LIN {X 0,Y 248.357,Z 469.454,A -85,B 0,C 180,E1 -18796.916,E2 -18796.916} C_VEL
LIN {X 0,Y 247.432,Z 473.592,A -85,B 0,C 180,E1 -18800.188,E2 -18800.188} C_VEL
LIN {X 0,Y 246.966,Z 476.493,A -85,B 0,C 180,E1 -18803.464,E2 -18803.464} C_VEL
LIN {X 0,Y 246.805,Z 478.221,A -85,B 0,C 180,E1 -18806.735,E2 -18806.735} C_VEL
LIN {X 0,Y 246.889,Z 478.812,A -85,B 0,C 180,E1 -18810,E2 -18810} C_VEL
LIN {X 0,Y 246.805,Z 478.208,A -85,B 0,C 180,E1 -18813.265,E2 -18813.265} C_VEL
LIN {X 0,Y 246.966,Z 476.463,A -85,B 0,C 180,E1 -18816.536,E2 -18816.536} C_VEL
LIN {X 0,Y 247.428,Z 473.551,A -85,B 0,C 180,E1 -18819.813,E2 -18819.813} C_VEL
LIN {X 0,Y 248.352,Z 469.403,A -85,B 0,C 180,E1 -18823.084,E2 -18823.084} C_VEL
LIN {X 0,Y 249.899,Z 463.909,A -85,B 0,C 180,E1 -18826.334,E2 -18826.334} C_VEL
LIN {X 0,Y 252.033,Z 456.92,A -85,B 0,C 180,E1 -18829.55,E2 -18829.55} C_VEL
LIN {X 0,Y 254.843,Z 448.224,A -85,B 0,C 180,E1 -18832.711,E2 -18832.711} C_VEL
LIN {X 0,Y 257.993,Z 438.986,A -85,B 0,C 180,E1 -18835.407,E2 -18835.407} C_VEL
LIN {X 0,Y 260.373,Z 431.227,A -85,B 0,C 180,E1 -18837.314,E2 -18837.314} C_VEL
LIN {X 0,Y 263.812,Z 420.385,A -85,B 0,C 180,E1 -18839.528,E2 -18839.528} C_VEL
LIN {X 0,Y 267.196,Z 408.548,A -85,B 0,C 180,E1 -18841.518,E2 -18841.518} C_VEL
LIN {X 0,Y 270.674,Z 395.599,A -85,B 0,C 180,E1 -18843.265,E2 -18843.265} C_VEL
LIN {X 0,Y 273.816,Z 381.642,A -85,B 0,C 180,E1 -18844.781,E2 -18844.781} C_VEL
LIN {X 0,Y 276.434,Z 367.299,A -85,B 0,C 180,E1 -18846.01,E2 -18846.01} C_VEL
LIN {X 0,Y 278.793,Z 352.325,A -85,B 0,C 180,E1 -18846.947,E2 -18846.947} C_VEL
LIN {X 0,Y 280.556,Z 336.654,A -85,B 0,C 180,E1 -18847.633,E2 -18847.633} C_VEL
LIN {X 0,Y 281.741,Z 316.789,A -85,B 0,C 180,E1 -18848.182,E2 -18848.182} C_VEL
LIN {X 0,Y 285.687,Z 232.335,A -85,B 0,C 180,E1 -18850.234,E2 -18850.234} C_VEL
LIN {X 0,Y 278.998,Z 217.135,A -85,B 0,C 180,E1 -18851.915,E2 -18851.915} C_VEL
LIN {X 0,Y 272.04,Z 203.261,A -85,B 0,C 180,E1 -18853.734,E2 -18853.734} C_VEL
LIN {X 0,Y 264.682,Z 190.304,A -85,B 0,C 180,E1 -18855.764,E2 -18855.764} C_VEL
LIN {X 0,Y 258.697,Z 180.792,A -85,B 0,C 180,E1 -18857.519,E2 -18857.519} C_VEL
LIN {X 0,Y 255.268,Z 175.543,A -85,B 0,C 180,E1 -18858.582,E2 -18858.582} C_VEL
LIN {X 0,Y 252.372,Z 171.249,A -85,B 0,C 180,E1 -18859.514,E2 -18859.514} C_VEL
LIN {X 0,Y 249.479,Z 166.762,A -85,B 0,C 180,E1 -18860.601,E2 -18860.601} C_VEL
LIN {X 0,Y 249.055,Z 165.14,A -85,B 0,C 180,E1 -18861.496,E2 -18861.496} C_VEL
LIN {X 0,Y 249.061,Z 165.021,A -85,B 0,C 180,E1 -18865.642,E2 -18865.642} C_VEL
LIN {X 0,Y 249.052,Z 165.043,A -85,B 0,C 180,E1 -18869.473,E2 -18869.473} C_VEL
LIN {X 0,Y 249.076,Z 165.066,A -85,B 0,C 180,E1 -18873.163,E2 -18873.163} C_VEL
LIN {X 0,Y 249.083,Z 165.081,A -85,B 0,C 180,E1 -18876.733,E2 -18876.733} C_VEL
LIN {X 0,Y 249.112,Z 165.064,A -85,B 0,C 180,E1 -18880.212,E2 -18880.212} C_VEL
LIN {X 0,Y 249.243,Z 165.041,A -85,B 0,C 180,E1 -18883.622,E2 -18883.622} C_VEL
LIN {X 0,Y 249.245,Z 165.05,A -85,B 0,C 180,E1 -18888.616,E2 -18888.616} C_VEL
LIN {X 0,Y 249.42,Z 165.025,A -85,B 0,C 180,E1 -18891.901,E2 -18891.901} C_VEL
LIN {X 0,Y 249.281,Z 165.035,A -85,B 0,C 180,E1 -18895.148,E2 -18895.148} C_VEL
LIN {X 0,Y 249.674,Z 164.998,A -85,B 0,C 180,E1 -18898.387,E2 -18898.387} C_VEL
LIN {X 0,Y 249.665,Z 164.984,A -85,B 0,C 180,E1 -18901.613,E2 -18901.613} C_VEL
LIN {X 0,Y 249.427,Z 165.032,A -85,B 0,C 180,E1 -18906.541,E2 -18906.541} C_VEL
LIN {X 0,Y 249.344,Z 165.03,A -85,B 0,C 180,E1 -18909.737,E2 -18909.737} C_VEL
LIN {X 0,Y 249.172,Z 165.046,A -85,B 0,C 180,E1 -18914.706,E2 -18914.706} C_VEL
LIN {X 0,Y 249.096,Z 165.075,A -85,B 0,C 180,E1 -18918.081,E2 -18918.081} C_VEL
LIN {X 0,Y 249.044,Z 165.074,A -85,B 0,C 180,E1 -18921.522,E2 -18921.522} C_VEL
LIN {X 0,Y 249.048,Z 165.066,A -85,B 0,C 180,E1 -18925.442,E2 -18925.442} C_VEL
LIN {X 0,Y 249.035,Z 165.064,A -85,B 0,C 180,E1 -18928.973,E2 -18928.973} C_VEL
LIN {X 0,Y 249.028,Z 165.016,A -85,B 0,C 180,E1 -18932.426,E2 -18932.426} C_VEL
LIN {X 0,Y 249.03,Z 165.093,A -85,B 0,C 180,E1 -18936.346,E2 -18936.346} C_VEL
LIN {X 0,Y 249.032,Z 165.261,A -85,B 0,C 180,E1 -18939.157,E2 -18939.157} C_VEL
LIN {X 0,Y 249.258,Z 166.289,A -85,B 0,C 180,E1 -18939.571,E2 -18939.571} C_VEL
LIN {X 0,Y 250.775,Z 168.943,A -85,B 0,C 180,E1 -18940.134,E2 -18940.134} C_VEL
LIN {X 0,Y 252.601,Z 170.697,A -85,B 0,C 180,E1 -18940.7,E2 -18940.7} C_VEL
LIN {X 0,Y 254.742,Z 174.012,A -85,B 0,C 180,E1 -18941.397,E2 -18941.397} C_VEL
LIN {X 0,Y 256.104,Z 175.59,A -85,B 0,C 180,E1 -18941.808,E2 -18941.808} C_VEL
LIN {X 0,Y 258.812,Z 179.338,A -85,B 0,C 180,E1 -18942.627,E2 -18942.627} C_VEL
LIN {X 0,Y 263.301,Z 186.225,A -85,B 0,C 180,E1 -18943.947,E2 -18943.947} C_VEL
LIN {X 0,Y 270.19,Z 197.804,A -85,B 0,C 180,E1 -18945.869,E2 -18945.869} C_VEL
LIN {X 0,Y 277.344,Z 211.184,A -85,B 0,C 180,E1 -18947.751,E2 -18947.751} C_VEL
LIN {X 0,Y 283.547,Z 224.507,A -85,B 0,C 180,E1 -18949.321,E2 -18949.321} C_VEL
LIN {X 0,Y 285.786,Z 229.616,A -85,B 0,C 180,E1 -18949.872,E2 -18949.872} C_VEL
LIN {X 0,Y 281.718,Z 316.592,A -85,B 0,C 180,E1 -18951.984,E2 -18951.984} C_VEL
LIN {X 0,Y 280.587,Z 333.873,A -85,B 0,C 180,E1 -18952.485,E2 -18952.485} C_VEL
LIN {X 0,Y 278.901,Z 349.072,A -85,B 0,C 180,E1 -18953.183,E2 -18953.183} C_VEL
LIN {X 0,Y 276.858,Z 362.663,A -85,B 0,C 180,E1 -18954.054,E2 -18954.054} C_VEL
LIN {X 0,Y 274.288,Z 376.81,A -85,B 0,C 180,E1 -18955.253,E2 -18955.253} C_VEL
LIN {X 0,Y 271.157,Z 391.075,A -85,B 0,C 180,E1 -18956.802,E2 -18956.802} C_VEL
LIN {X 0,Y 267.701,Z 404.046,A -85,B 0,C 180,E1 -18958.548,E2 -18958.548} C_VEL
LIN {X 0,Y 264.306,Z 415.889,A -85,B 0,C 180,E1 -18960.533,E2 -18960.533} C_VEL
LIN {X 0,Y 260.969,Z 426.728,A -85,B 0,C 180,E1 -18962.754,E2 -18962.754} C_VEL
LIN {X 0,Y 258.082,Z 435.921,A -85,B 0,C 180,E1 -18965.033,E2 -18965.033} C_VEL
LIN {X 0,Y 255.039,Z 444.915,A -85,B 0,C 180,E1 -18967.734,E2 -18967.734} C_VEL
LIN {X 0,Y 252.502,Z 452.369,A -85,B 0,C 180,E1 -18970.488,E2 -18970.488} C_VEL
LIN {X 0,Y 250.312,Z 459.336,A -85,B 0,C 180,E1 -18973.694,E2 -18973.694} C_VEL
LIN {X 0,Y 248.66,Z 464.811,A -85,B 0,C 180,E1 -18976.932,E2 -18976.932} C_VEL
LIN {X 0,Y 247.663,Z 468.943,A -85,B 0,C 180,E1 -18980.197,E2 -18980.197} C_VEL
LIN {X 0,Y 247.075,Z 471.845,A -85,B 0,C 180,E1 -18983.467,E2 -18983.467} C_VEL
LIN {X 0,Y 246.873,Z 473.588,A -85,B 0,C 180,E1 -18986.736,E2 -18986.736} C_VEL
LIN {X 0,Y 246.892,Z 474.196,A -85,B 0,C 180,E1 -18990,E2 -18990} C_VEL
LIN {X 0,Y 246.871,Z 473.628,A -85,B 0,C 180,E1 -18993.264,E2 -18993.264} C_VEL
LIN {X 0,Y 247.068,Z 471.936,A -85,B 0,C 180,E1 -18996.534,E2 -18996.534} C_VEL
LIN {X 0,Y 247.647,Z 469.082,A -85,B 0,C 180,E1 -18999.804,E2 -18999.804} C_VEL
LIN {X 0,Y 248.635,Z 464.997,A -85,B 0,C 180,E1 -19003.07,E2 -19003.07} C_VEL
LIN {X 0,Y 250.273,Z 459.581,A -85,B 0,C 180,E1 -19006.309,E2 -19006.309} C_VEL
LIN {X 0,Y 252.478,Z 452.682,A -85,B 0,C 180,E1 -19009.514,E2 -19009.514} C_VEL
LIN {X 0,Y 255.366,Z 444.071,A -85,B 0,C 180,E1 -19012.662,E2 -19012.662} C_VEL
LIN {X 0,Y 258.04,Z 436.329,A -85,B 0,C 180,E1 -19014.971,E2 -19014.971} C_VEL
LIN {X 0,Y 261.403,Z 425.595,A -85,B 0,C 180,E1 -19017.631,E2 -19017.631} C_VEL
LIN {X 0,Y 265.139,Z 413.53,A -85,B 0,C 180,E1 -19020.021,E2 -19020.021} C_VEL
LIN {X 0,Y 268.63,Z 401.209,A -85,B 0,C 180,E1 -19021.991,E2 -19021.991} C_VEL
LIN {X 0,Y 272.023,Z 387.612,A -85,B 0,C 180,E1 -19023.744,E2 -19023.744} C_VEL
LIN {X 0,Y 274.945,Z 374.176,A -85,B 0,C 180,E1 -19025.118,E2 -19025.118} C_VEL
LIN {X 0,Y 277.462,Z 359.466,A -85,B 0,C 180,E1 -19026.305,E2 -19026.305} C_VEL
LIN {X 0,Y 279.677,Z 343.923,A -85,B 0,C 180,E1 -19027.205,E2 -19027.205} C_VEL
LIN {X 0,Y 281.176,Z 328.456,A -85,B 0,C 180,E1 -19027.819,E2 -19027.819} C_VEL
LIN {X 0,Y 285.935,Z 229.905,A -85,B 0,C 180,E1 -19030.23,E2 -19030.23} C_VEL
LIN {X 0,Y 279.759,Z 216.163,A -85,B 0,C 180,E1 -19031.772,E2 -19031.772} C_VEL
LIN {X 0,Y 273.11,Z 203.043,A -85,B 0,C 180,E1 -19033.497,E2 -19033.497} C_VEL
LIN {X 0,Y 264.585,Z 188.119,A -85,B 0,C 180,E1 -19035.845,E2 -19035.845} C_VEL
LIN {X 0,Y 258.741,Z 179.263,A -85,B 0,C 180,E1 -19037.552,E2 -19037.552} C_VEL
LIN {X 0,Y 256.012,Z 175.393,A -85,B 0,C 180,E1 -19038.385,E2 -19038.385} C_VEL
LIN {X 0,Y 253.144,Z 171.8,A -85,B 0,C 180,E1 -19039.275,E2 -19039.275} C_VEL
LIN {X 0,Y 252.157,Z 170.153,A -85,B 0,C 180,E1 -19039.608,E2 -19039.608} C_VEL
LIN {X 0,Y 250.029,Z 167.934,A -85,B 0,C 180,E1 -19040.283,E2 -19040.283} C_VEL
LIN {X 0,Y 249.097,Z 165.61,A -85,B 0,C 180,E1 -19040.79,E2 -19040.79} C_VEL
LIN {X 0,Y 249.017,Z 165.181,A -85,B 0,C 180,E1 -19041.1,E2 -19041.1} C_VEL
LIN {X 0,Y 249.044,Z 165.038,A -85,B 0,C 180,E1 -19045.639,E2 -19045.639} C_VEL
LIN {X 0,Y 249.002,Z 165.03,A -85,B 0,C 180,E1 -19049.466,E2 -19049.466} C_VEL
LIN {X 0,Y 249.026,Z 165.083,A -85,B 0,C 180,E1 -19053.157,E2 -19053.157} C_VEL
LIN {X 0,Y 249.008,Z 165.086,A -85,B 0,C 180,E1 -19056.725,E2 -19056.725} C_VEL
LIN {X 0,Y 249.047,Z 165.064,A -85,B 0,C 180,E1 -19060.206,E2 -19060.206} C_VEL
LIN {X 0,Y 249.095,Z 165.071,A -85,B 0,C 180,E1 -19062.51,E2 -19062.51} C_VEL
LIN {X 0,Y 248.463,Z 165.153,A -85,B 0,C 180,E1 -19063.86,E2 -19063.86} C_VEL
LIN {X 0,Y 245.618,Z 165.507,A -85,B 0,C 180,E1 -19066.061,E2 -19066.061} C_VEL
LIN {X 0,Y 243.23,Z 165.808,A -85,B 0,C 180,E1 -19067.854,E2 -19067.854} C_VEL
LIN {X 0,Y 242.277,Z 165.926,A -85,B 0,C 180,E1 -19069.246,E2 -19069.246} C_VEL
LIN {X 0,Y 242.239,Z 165.92,A -85,B 0,C 180,E1 -19069.716,E2 -19069.716} C_VEL
LIN {X 0,Y 242.402,Z 165.903,A -85,B 0,C 180,E1 -19073.34,E2 -19073.34} C_VEL
LIN {X 0,Y 242.624,Z 165.86,A -85,B 0,C 180,E1 -19078.34,E2 -19078.34} C_VEL
LIN {X 0,Y 242.632,Z 165.874,A -85,B 0,C 180,E1 -19081.66,E2 -19081.66} C_VEL
LIN {X 0,Y 242.402,Z 165.914,A -85,B 0,C 180,E1 -19086.66,E2 -19086.66} C_VEL
LIN {X 0,Y 242.269,Z 165.905,A -85,B 0,C 180,E1 -19090.023,E2 -19090.023} C_VEL
LIN {X 0,Y 242.168,Z 165.92,A -85,B 0,C 180,E1 -19095.141,E2 -19095.141} C_VEL
LIN {X 0,Y 242.073,Z 165.956,A -85,B 0,C 180,E1 -19098.624,E2 -19098.624} C_VEL
LIN {X 0,Y 242.008,Z 165.948,A -85,B 0,C 180,E1 -19102.18,E2 -19102.18} C_VEL
LIN {X 0,Y 242.068,Z 165.936,A -85,B 0,C 180,E1 -19105.838,E2 -19105.838} C_VEL
LIN {X 0,Y 242.032,Z 165.938,A -85,B 0,C 180,E1 -19109.58,E2 -19109.58} C_VEL
LIN {X 0,Y 241.981,Z 165.895,A -85,B 0,C 180,E1 -19113.492,E2 -19113.492} C_VEL
LIN {X 0,Y 242.019,Z 166.117,A -85,B 0,C 180,E1 -19116.792,E2 -19116.792} C_VEL
LIN {X 0,Y 242.243,Z 167.162,A -85,B 0,C 180,E1 -19117.274,E2 -19117.274} C_VEL
LIN {X 0,Y 243.897,Z 169.988,A -85,B 0,C 180,E1 -19117.957,E2 -19117.957} C_VEL
LIN {X 0,Y 246.212,Z 172.655,A -85,B 0,C 180,E1 -19118.763,E2 -19118.763} C_VEL
LIN {X 0,Y 251.482,Z 180.476,A -85,B 0,C 180,E1 -19120.57,E2 -19120.57} C_VEL
LIN {X 0,Y 256.805,Z 188.703,A -85,B 0,C 180,E1 -19122.272,E2 -19122.272} C_VEL
LIN {X 0,Y 264.449,Z 201.618,A -85,B 0,C 180,E1 -19124.552,E2 -19124.552} C_VEL
LIN {X 0,Y 271.551,Z 215.178,A -85,B 0,C 180,E1 -19126.538,E2 -19126.538} C_VEL
LIN {X 0,Y 278.07,Z 229.34,A -85,B 0,C 180,E1 -19128.277,E2 -19128.277} C_VEL
LIN {X 0,Y 280.293,Z 234.633,A -85,B 0,C 180,E1 -19128.857,E2 -19128.857} C_VEL
LIN {X 0,Y 276.265,Z 318.148,A -85,B 0,C 180,E1 -19130.919,E2 -19130.919} C_VEL
LIN {X 0,Y 274.995,Z 337.484,A -85,B 0,C 180,E1 -19131.468,E2 -19131.468} C_VEL
LIN {X 0,Y 273.172,Z 352.844,A -85,B 0,C 180,E1 -19132.161,E2 -19132.161} C_VEL
LIN {X 0,Y 270.766,Z 367.673,A -85,B 0,C 180,E1 -19133.113,E2 -19133.113} C_VEL
LIN {X 0,Y 268.109,Z 381.58,A -85,B 0,C 180,E1 -19134.322,E2 -19134.322} C_VEL
LIN {X 0,Y 264.756,Z 395.836,A -85,B 0,C 180,E1 -19135.895,E2 -19135.895} C_VEL
LIN {X 0,Y 261.181,Z 408.699,A -85,B 0,C 180,E1 -19137.669,E2 -19137.669} C_VEL
LIN {X 0,Y 257.616,Z 420.502,A -85,B 0,C 180,E1 -19139.689,E2 -19139.689} C_VEL
LIN {X 0,Y 254.101,Z 431.316,A -85,B 0,C 180,E1 -19141.953,E2 -19141.953} C_VEL
LIN {X 0,Y 251.09,Z 440.49,A -85,B 0,C 180,E1 -19144.288,E2 -19144.288} C_VEL
LIN {X 0,Y 247.865,Z 449.488,A -85,B 0,C 180,E1 -19147.053,E2 -19147.053} C_VEL
LIN {X 0,Y 245.287,Z 456.953,A -85,B 0,C 180,E1 -19149.89,E2 -19149.89} C_VEL
LIN {X 0,Y 243.073,Z 463.916,A -85,B 0,C 180,E1 -19153.194,E2 -19153.194} C_VEL
LIN {X 0,Y 241.414,Z 469.389,A -85,B 0,C 180,E1 -19156.532,E2 -19156.532} C_VEL
LIN {X 0,Y 240.398,Z 473.526,A -85,B 0,C 180,E1 -19159.897,E2 -19159.897} C_VEL
LIN {X 0,Y 239.889,Z 476.426,A -85,B 0,C 180,E1 -19163.27,E2 -19163.27} C_VEL
LIN {X 0,Y 239.713,Z 478.155,A -85,B 0,C 180,E1 -19166.638,E2 -19166.638} C_VEL
LIN {X 0,Y 239.801,Z 478.746,A -85,B 0,C 180,E1 -19170,E2 -19170} C_VEL
LIN {X 0,Y 239.714,Z 478.141,A -85,B 0,C 180,E1 -19173.361,E2 -19173.361} C_VEL
LIN {X 0,Y 239.888,Z 476.396,A -85,B 0,C 180,E1 -19176.73,E2 -19176.73} C_VEL
LIN {X 0,Y 240.393,Z 473.483,A -85,B 0,C 180,E1 -19180.103,E2 -19180.103} C_VEL
LIN {X 0,Y 241.409,Z 469.335,A -85,B 0,C 180,E1 -19183.468,E2 -19183.468} C_VEL
LIN {X 0,Y 243.039,Z 463.841,A -85,B 0,C 180,E1 -19186.808,E2 -19186.808} C_VEL
LIN {X 0,Y 245.285,Z 456.852,A -85,B 0,C 180,E1 -19190.11,E2 -19190.11} C_VEL
LIN {X 0,Y 248.248,Z 448.155,A -85,B 0,C 180,E1 -19193.35,E2 -19193.35} C_VEL
LIN {X 0,Y 251.07,Z 440.361,A -85,B 0,C 180,E1 -19195.714,E2 -19195.714} C_VEL
LIN {X 0,Y 253.544,Z 432.629,A -85,B 0,C 180,E1 -19197.708,E2 -19197.708} C_VEL
LIN {X 0,Y 257.018,Z 422.268,A -85,B 0,C 180,E1 -19199.936,E2 -19199.936} C_VEL
LIN {X 0,Y 260.493,Z 410.827,A -85,B 0,C 180,E1 -19201.97,E2 -19201.97} C_VEL
LIN {X 0,Y 264.008,Z 398.385,A -85,B 0,C 180,E1 -19203.759,E2 -19203.759} C_VEL
LIN {X 0,Y 267.365,Z 384.748,A -85,B 0,C 180,E1 -19205.331,E2 -19205.331} C_VEL
LIN {X 0,Y 270.141,Z 370.612,A -85,B 0,C 180,E1 -19206.637,E2 -19206.637} C_VEL
LIN {X 0,Y 272.682,Z 356.046,A -85,B 0,C 180,E1 -19207.627,E2 -19207.627} C_VEL
LIN {X 0,Y 274.531,Z 341.075,A -85,B 0,C 180,E1 -19208.375,E2 -19208.375} C_VEL
LIN {X 0,Y 275.742,Z 325.627,A -85,B 0,C 180,E1 -19208.876,E2 -19208.876} C_VEL
LIN {X 0,Y 280.23,Z 235.291,A -85,B 0,C 180,E1 -19211.083,E2 -19211.083} C_VEL
LIN {X 0,Y 279.636,Z 233.207,A -85,B 0,C 180,E1 -19211.258,E2 -19211.258} C_VEL
LIN {X 0,Y 273.037,Z 218.349,A -85,B 0,C 180,E1 -19213.002,E2 -19213.002} C_VEL
LIN {X 0,Y 266.227,Z 204.956,A -85,B 0,C 180,E1 -19214.876,E2 -19214.876} C_VEL
LIN {X 0,Y 258.939,Z 192.192,A -85,B 0,C 180,E1 -19217.006,E2 -19217.006} C_VEL
LIN {X 0,Y 251.789,Z 180.975,A -85,B 0,C 180,E1 -19219.252,E2 -19219.252} C_VEL
LIN {X 0,Y 246.85,Z 173.669,A -85,B 0,C 180,E1 -19220.925,E2 -19220.925} C_VEL
LIN {X 0,Y 244.436,Z 170.507,A -85,B 0,C 180,E1 -19221.772,E2 -19221.772} C_VEL
LIN {X 0,Y 242.548,Z 167.907,A -85,B 0,C 180,E1 -19222.48,E2 -19222.48} C_VEL
LIN {X 0,Y 242.098,Z 166.534,A -85,B 0,C 180,E1 -19222.831,E2 -19222.831} C_VEL
LIN {X 0,Y 242.029,Z 165.989,A -85,B 0,C 180,E1 -19223.469,E2 -19223.469} C_VEL
LIN {X 0,Y 241.996,Z 165.892,A -85,B 0,C 180,E1 -19227.375,E2 -19227.375} C_VEL
LIN {X 0,Y 242.038,Z 165.945,A -85,B 0,C 180,E1 -19230.587,E2 -19230.587} C_VEL
LIN {X 0,Y 242.068,Z 165.936,A -85,B 0,C 180,E1 -19234.183,E2 -19234.183} C_VEL
LIN {X 0,Y 242.054,Z 165.937,A -85,B 0,C 180,E1 -19238.297,E2 -19238.297} C_VEL
LIN {X 0,Y 242.164,Z 165.926,A -85,B 0,C 180,E1 -19243.278,E2 -19243.278} C_VEL
LIN {X 0,Y 242.181,Z 165.934,A -85,B 0,C 180,E1 -19248.28,E2 -19248.28} C_VEL
LIN {X 0,Y 242.374,Z 165.898,A -85,B 0,C 180,E1 -19251.664,E2 -19251.664} C_VEL
LIN {X 0,Y 242.241,Z 165.913,A -85,B 0,C 180,E1 -19255.007,E2 -19255.007} C_VEL
LIN {X 0,Y 242.634,Z 165.873,A -85,B 0,C 180,E1 -19258.34,E2 -19258.34} C_VEL
LIN {X 0,Y 242.624,Z 165.86,A -85,B 0,C 180,E1 -19261.66,E2 -19261.66} C_VEL
LIN {X 0,Y 242.402,Z 165.904,A -85,B 0,C 180,E1 -19266.66,E2 -19266.66} C_VEL
LIN {X 0,Y 242.268,Z 165.914,A -85,B 0,C 180,E1 -19270.024,E2 -19270.024} C_VEL
LIN {X 0,Y 242.127,Z 165.925,A -85,B 0,C 180,E1 -19275.144,E2 -19275.144} C_VEL
LIN {X 0,Y 242.032,Z 165.946,A -85,B 0,C 180,E1 -19278.628,E2 -19278.628} C_VEL
LIN {X 0,Y 241.974,Z 165.965,A -85,B 0,C 180,E1 -19282.184,E2 -19282.184} C_VEL
LIN {X 0,Y 241.988,Z 165.947,A -85,B 0,C 180,E1 -19285.826,E2 -19285.826} C_VEL
LIN {X 0,Y 241.968,Z 165.925,A -85,B 0,C 180,E1 -19289.589,E2 -19289.589} C_VEL
LIN {X 0,Y 241.98,Z 165.899,A -85,B 0,C 180,E1 -19293.493,E2 -19293.493} C_VEL
LIN {X 0,Y 241.997,Z 166.189,A -85,B 0,C 180,E1 -19297.188,E2 -19297.188} C_VEL
LIN {X 0,Y 242.322,Z 167.358,A -85,B 0,C 180,E1 -19297.599,E2 -19297.599} C_VEL
LIN {X 0,Y 243.904,Z 169.99,A -85,B 0,C 180,E1 -19298.222,E2 -19298.222} C_VEL
LIN {X 0,Y 245.675,Z 171.559,A -85,B 0,C 180,E1 -19298.817,E2 -19298.817} C_VEL
LIN {X 0,Y 247.691,Z 174.793,A -85,B 0,C 180,E1 -19299.54,E2 -19299.54} C_VEL
LIN {X 0,Y 249.386,Z 176.695,A -85,B 0,C 180,E1 -19300.094,E2 -19300.094} C_VEL
LIN {X 0,Y 252.129,Z 180.413,A -85,B 0,C 180,E1 -19300.99,E2 -19300.99} C_VEL
LIN {X 0,Y 258.645,Z 189.867,A -85,B 0,C 180,E1 -19303.009,E2 -19303.009} C_VEL
LIN {X 0,Y 266.274,Z 202.948,A -85,B 0,C 180,E1 -19305.235,E2 -19305.235} C_VEL
LIN {X 0,Y 273.18,Z 216.193,A -85,B 0,C 180,E1 -19307.127,E2 -19307.127} C_VEL
LIN {X 0,Y 279.304,Z 229.585,A -85,B 0,C 180,E1 -19308.737,E2 -19308.737} C_VEL
LIN {X 0,Y 280.283,Z 231.882,A -85,B 0,C 180,E1 -19308.989,E2 -19308.989} C_VEL
LIN {X 0,Y 275.984,Z 320.258,A -85,B 0,C 180,E1 -19311.165,E2 -19311.165} C_VEL
LIN {X 0,Y 274.806,Z 336.236,A -85,B 0,C 180,E1 -19311.671,E2 -19311.671} C_VEL
LIN {X 0,Y 272.958,Z 351.434,A -85,B 0,C 180,E1 -19312.418,E2 -19312.418} C_VEL
LIN {X 0,Y 270.761,Z 364.991,A -85,B 0,C 180,E1 -19313.345,E2 -19313.345} C_VEL
LIN {X 0,Y 268.153,Z 378.46,A -85,B 0,C 180,E1 -19314.546,E2 -19314.546} C_VEL
LIN {X 0,Y 264.835,Z 392.572,A -85,B 0,C 180,E1 -19316.132,E2 -19316.132} C_VEL
LIN {X 0,Y 261.314,Z 405.288,A -85,B 0,C 180,E1 -19317.915,E2 -19317.915} C_VEL
LIN {X 0,Y 258.14,Z 415.959,A -85,B 0,C 180,E1 -19319.757,E2 -19319.757} C_VEL
LIN {X 0,Y 254.558,Z 427.003,A -85,B 0,C 180,E1 -19322.065,E2 -19322.065} C_VEL
LIN {X 0,Y 251.641,Z 435.99,A -85,B 0,C 180,E1 -19324.349,E2 -19324.349} C_VEL
LIN {X 0,Y 248.436,Z 444.984,A -85,B 0,C 180,E1 -19327.109,E2 -19327.109} C_VEL
LIN {X 0,Y 245.766,Z 452.438,A -85,B 0,C 180,E1 -19329.931,E2 -19329.931} C_VEL
LIN {X 0,Y 243.442,Z 459.405,A -85,B 0,C 180,E1 -19333.22,E2 -19333.22} C_VEL
LIN {X 0,Y 241.706,Z 464.879,A -85,B 0,C 180,E1 -19336.549,E2 -19336.549} C_VEL
LIN {X 0,Y 240.641,Z 469.01,A -85,B 0,C 180,E1 -19339.908,E2 -19339.908} C_VEL
LIN {X 0,Y 240.02,Z 471.912,A -85,B 0,C 180,E1 -19343.274,E2 -19343.274} C_VEL
LIN {X 0,Y 239.78,Z 473.655,A -85,B 0,C 180,E1 -19346.639,E2 -19346.639} C_VEL
LIN {X 0,Y 239.805,Z 474.262,A -85,B 0,C 180,E1 -19350,E2 -19350} C_VEL
LIN {X 0,Y 239.778,Z 473.694,A -85,B 0,C 180,E1 -19353.361,E2 -19353.361} C_VEL
LIN {X 0,Y 239.991,Z 472.002,A -85,B 0,C 180,E1 -19356.727,E2 -19356.727} C_VEL
LIN {X 0,Y 240.625,Z 469.148,A -85,B 0,C 180,E1 -19360.093,E2 -19360.093} C_VEL
LIN {X 0,Y 241.68,Z 465.063,A -85,B 0,C 180,E1 -19363.453,E2 -19363.453} C_VEL
LIN {X 0,Y 243.406,Z 459.647,A -85,B 0,C 180,E1 -19366.782,E2 -19366.782} C_VEL
LIN {X 0,Y 245.725,Z 452.747,A -85,B 0,C 180,E1 -19370.073,E2 -19370.073} C_VEL
LIN {X 0,Y 248.773,Z 444.136,A -85,B 0,C 180,E1 -19373.298,E2 -19373.298} C_VEL
LIN {X 0,Y 251.594,Z 436.393,A -85,B 0,C 180,E1 -19375.657,E2 -19375.657} C_VEL
LIN {X 0,Y 254.539,Z 427.283,A -85,B 0,C 180,E1 -19377.994,E2 -19377.994} C_VEL
LIN {X 0,Y 258.047,Z 416.534,A -85,B 0,C 180,E1 -19380.255,E2 -19380.255} C_VEL
LIN {X 0,Y 261.573,Z 404.801,A -85,B 0,C 180,E1 -19382.277,E2 -19382.277} C_VEL
LIN {X 0,Y 265.08,Z 391.987,A -85,B 0,C 180,E1 -19384.062,E2 -19384.062} C_VEL
LIN {X 0,Y 268.368,Z 377.986,A -85,B 0,C 180,E1 -19385.621,E2 -19385.621} C_VEL
LIN {X 0,Y 270.991,Z 364.061,A -85,B 0,C 180,E1 -19386.851,E2 -19386.851} C_VEL
LIN {X 0,Y 273.304,Z 349.398,A -85,B 0,C 180,E1 -19387.817,E2 -19387.817} C_VEL
LIN {X 0,Y 275.096,Z 334.339,A -85,B 0,C 180,E1 -19388.515,E2 -19388.515} C_VEL
LIN {X 0,Y 276.242,Z 317.3,A -85,B 0,C 180,E1 -19389.026,E2 -19389.026} C_VEL
LIN {X 0,Y 280.441,Z 232.086,A -85,B 0,C 180,E1 -19391.115,E2 -19391.115} C_VEL
LIN {X 0,Y 273.936,Z 217.64,A -85,B 0,C 180,E1 -19392.819,E2 -19392.819} C_VEL
LIN {X 0,Y 267.329,Z 204.843,A -85,B 0,C 180,E1 -19394.619,E2 -19394.619} C_VEL
LIN {X 0,Y 260.233,Z 192.503,A -85,B 0,C 180,E1 -19396.669,E2 -19396.669} C_VEL
LIN {X 0,Y 255.358,Z 184.878,A -85,B 0,C 180,E1 -19398.157,E2 -19398.157} C_VEL
LIN {X 0,Y 251.658,Z 179.888,A -85,B 0,C 180,E1 -19399.322,E2 -19399.322} C_VEL
LIN {X 0,Y 248.577,Z 175.704,A -85,B 0,C 180,E1 -19400.342,E2 -19400.342} C_VEL
LIN {X 0,Y 246.139,Z 172.52,A -85,B 0,C 180,E1 -19401.177,E2 -19401.177} C_VEL
LIN {X 0,Y 245.214,Z 171.076,A -85,B 0,C 180,E1 -19401.514,E2 -19401.514} C_VEL
LIN {X 0,Y 242.985,Z 168.8,A -85,B 0,C 180,E1 -19402.289,E2 -19402.289} C_VEL
LIN {X 0,Y 242.069,Z 166.475,A -85,B 0,C 180,E1 -19402.825,E2 -19402.825} C_VEL
LIN {X 0,Y 241.984,Z 166.006,A -85,B 0,C 180,E1 -19403.201,E2 -19403.201} C_VEL
LIN {X 0,Y 241.989,Z 165.892,A -85,B 0,C 180,E1 -19407.377,E2 -19407.377} C_VEL
LIN {X 0,Y 241.977,Z 165.925,A -85,B 0,C 180,E1 -19410.613,E2 -19410.613} C_VEL
LIN {X 0,Y 241.997,Z 165.946,A -85,B 0,C 180,E1 -19414.197,E2 -19414.197} C_VEL
LIN {X 0,Y 241.987,Z 165.956,A -85,B 0,C 180,E1 -19418.337,E2 -19418.337} C_VEL
LIN {X 0,Y 242.115,Z 165.947,A -85,B 0,C 180,E1 -19423.318,E2 -19423.318} C_VEL
LIN {X 0,Y 242.168,Z 165.945,A -85,B 0,C 180,E1 -19428.279,E2 -19428.279} C_VEL
LIN {X 0,Y 242.239,Z 165.92,A -85,B 0,C 180,E1 -19429.716,E2 -19429.716} C_VEL
LIN {X 0,Y 241.648,Z 165.992,A -85,B 0,C 180,E1 -19431.104,E2 -19431.104} C_VEL
LIN {X 0,Y 238.752,Z 166.357,A -85,B 0,C 180,E1 -19433.365,E2 -19433.365} C_VEL
LIN {X 0,Y 236.311,Z 166.668,A -85,B 0,C 180,E1 -19435.21,E2 -19435.21} C_VEL
LIN {X 0,Y 235.369,Z 166.766,A -85,B 0,C 180,E1 -19436.643,E2 -19436.643} C_VEL
LIN {X 0,Y 235.353,Z 166.764,A -85,B 0,C 180,E1 -19437.128,E2 -19437.128} C_VEL
LIN {X 0,Y 235.641,Z 166.75,A -85,B 0,C 180,E1 -19440,E2 -19440} C_VEL
LIN {X 0,Y 235.591,Z 166.749,A -85,B 0,C 180,E1 -19441.709,E2 -19441.709} C_VEL
LIN {X 0,Y 235.353,Z 166.792,A -85,B 0,C 180,E1 -19446.86,E2 -19446.86} C_VEL
LIN {X 0,Y 235.216,Z 166.784,A -85,B 0,C 180,E1 -19450.327,E2 -19450.327} C_VEL
LIN {X 0,Y 235.115,Z 166.797,A -85,B 0,C 180,E1 -19455.606,E2 -19455.606} C_VEL
LIN {X 0,Y 235.009,Z 166.827,A -85,B 0,C 180,E1 -19459.205,E2 -19459.205} C_VEL
LIN {X 0,Y 234.954,Z 166.835,A -85,B 0,C 180,E1 -19462.883,E2 -19462.883} C_VEL
LIN {X 0,Y 234.971,Z 166.821,A -85,B 0,C 180,E1 -19466.657,E2 -19466.657} C_VEL
LIN {X 0,Y 234.932,Z 166.795,A -85,B 0,C 180,E1 -19470.567,E2 -19470.567} C_VEL
LIN {X 0,Y 234.93,Z 166.903,A -85,B 0,C 180,E1 -19474.426,E2 -19474.426} C_VEL
LIN {X 0,Y 235.123,Z 167.742,A -85,B 0,C 180,E1 -19474.942,E2 -19474.942} C_VEL
LIN {X 0,Y 236.523,Z 170.439,A -85,B 0,C 180,E1 -19475.632,E2 -19475.632} C_VEL
LIN {X 0,Y 238.958,Z 172.789,A -85,B 0,C 180,E1 -19476.553,E2 -19476.553} C_VEL
LIN {X 0,Y 241.148,Z 176.081,A -85,B 0,C 180,E1 -19477.407,E2 -19477.407} C_VEL
LIN {X 0,Y 243.323,Z 178.871,A -85,B 0,C 180,E1 -19478.201,E2 -19478.201} C_VEL
LIN {X 0,Y 249.864,Z 188.597,A -85,B 0,C 180,E1 -19480.489,E2 -19480.489} C_VEL
LIN {X 0,Y 258.016,Z 202.128,A -85,B 0,C 180,E1 -19483.105,E2 -19483.105} C_VEL
LIN {X 0,Y 265.681,Z 216.498,A -85,B 0,C 180,E1 -19485.377,E2 -19485.377} C_VEL
LIN {X 0,Y 272.909,Z 232.174,A -85,B 0,C 180,E1 -19487.405,E2 -19487.405} C_VEL
LIN {X 0,Y 274.928,Z 237.032,A -85,B 0,C 180,E1 -19487.957,E2 -19487.957} C_VEL
LIN {X 0,Y 270.002,Z 331.315,A -85,B 0,C 180,E1 -19490.317,E2 -19490.317} C_VEL
LIN {X 0,Y 268.537,Z 346.332,A -85,B 0,C 180,E1 -19490.908,E2 -19490.908} C_VEL
LIN {X 0,Y 266.404,Z 360.422,A -85,B 0,C 180,E1 -19491.687,E2 -19491.687} C_VEL
LIN {X 0,Y 263.871,Z 373.981,A -85,B 0,C 180,E1 -19492.705,E2 -19492.705} C_VEL
LIN {X 0,Y 260.839,Z 388.062,A -85,B 0,C 180,E1 -19494.099,E2 -19494.099} C_VEL
LIN {X 0,Y 257.37,Z 401.208,A -85,B 0,C 180,E1 -19495.722,E2 -19495.722} C_VEL
LIN {X 0,Y 253.439,Z 414.263,A -85,B 0,C 180,E1 -19497.736,E2 -19497.736} C_VEL
LIN {X 0,Y 249.557,Z 426.077,A -85,B 0,C 180,E1 -19500.008,E2 -19500.008} C_VEL
LIN {X 0,Y 245.953,Z 436.539,A -85,B 0,C 180,E1 -19502.494,E2 -19502.494} C_VEL
LIN {X 0,Y 242.687,Z 445.744,A -85,B 0,C 180,E1 -19505.171,E2 -19505.171} C_VEL
LIN {X 0,Y 239.686,Z 453.857,A -85,B 0,C 180,E1 -19508.047,E2 -19508.047} C_VEL
LIN {X 0,Y 237.264,Z 460.567,A -85,B 0,C 180,E1 -19510.984,E2 -19510.984} C_VEL
LIN {X 0,Y 235.276,Z 466.761,A -85,B 0,C 180,E1 -19514.405,E2 -19514.405} C_VEL
LIN {X 0,Y 233.807,Z 471.551,A -85,B 0,C 180,E1 -19517.853,E2 -19517.853} C_VEL
LIN {X 0,Y 233.035,Z 475.06,A -85,B 0,C 180,E1 -19521.327,E2 -19521.327} C_VEL
LIN {X 0,Y 232.686,Z 477.368,A -85,B 0,C 180,E1 -19524.801,E2 -19524.801} C_VEL
LIN {X 0,Y 232.644,Z 478.527,A -85,B 0,C 180,E1 -19528.269,E2 -19528.269} C_VEL
LIN {X 0,Y 232.715,Z 478.679,A -85,B 0,C 180,E1 -19530,E2 -19530} C_VEL
LIN {X 0,Y 232.625,Z 478.075,A -85,B 0,C 180,E1 -19533.464,E2 -19533.464} C_VEL
LIN {X 0,Y 232.807,Z 476.329,A -85,B 0,C 180,E1 -19536.935,E2 -19536.935} C_VEL
LIN {X 0,Y 233.372,Z 473.416,A -85,B 0,C 180,E1 -19540.41,E2 -19540.41} C_VEL
LIN {X 0,Y 234.475,Z 469.268,A -85,B 0,C 180,E1 -19543.874,E2 -19543.874} C_VEL
LIN {X 0,Y 236.17,Z 463.773,A -85,B 0,C 180,E1 -19547.312,E2 -19547.312} C_VEL
LIN {X 0,Y 238.568,Z 456.783,A -85,B 0,C 180,E1 -19550.702,E2 -19550.702} C_VEL
LIN {X 0,Y 241.686,Z 448.086,A -85,B 0,C 180,E1 -19554.023,E2 -19554.023} C_VEL
LIN {X 0,Y 244.632,Z 440.292,A -85,B 0,C 180,E1 -19556.442,E2 -19556.442} C_VEL
LIN {X 0,Y 247.186,Z 432.742,A -85,B 0,C 180,E1 -19558.433,E2 -19558.433} C_VEL
LIN {X 0,Y 250.853,Z 422.199,A -85,B 0,C 180,E1 -19560.75,E2 -19560.75} C_VEL
LIN {X 0,Y 254.445,Z 410.756,A -85,B 0,C 180,E1 -19562.824,E2 -19562.824} C_VEL
LIN {X 0,Y 258.124,Z 398.314,A -85,B 0,C 180,E1 -19564.637,E2 -19564.637} C_VEL
LIN {X 0,Y 261.583,Z 384.676,A -85,B 0,C 180,E1 -19566.234,E2 -19566.234} C_VEL
LIN {X 0,Y 264.457,Z 370.538,A -85,B 0,C 180,E1 -19567.558,E2 -19567.558} C_VEL
LIN {X 0,Y 267.16,Z 355.224,A -85,B 0,C 180,E1 -19568.605,E2 -19568.605} C_VEL
LIN {X 0,Y 269.108,Z 339.919,A -85,B 0,C 180,E1 -19569.355,E2 -19569.355} C_VEL
LIN {X 0,Y 270.361,Z 323.771,A -85,B 0,C 180,E1 -19569.862,E2 -19569.862} C_VEL
LIN {X 0,Y 274.755,Z 236.769,A -85,B 0,C 180,E1 -19572.032,E2 -19572.032} C_VEL
LIN {X 0,Y 268.537,Z 222.554,A -85,B 0,C 180,E1 -19573.748,E2 -19573.748} C_VEL
LIN {X 0,Y 261.701,Z 208.95,A -85,B 0,C 180,E1 -19575.715,E2 -19575.715} C_VEL
LIN {X 0,Y 254.909,Z 196.946,A -85,B 0,C 180,E1 -19577.788,E2 -19577.788} C_VEL
LIN {X 0,Y 248.065,Z 185.969,A -85,B 0,C 180,E1 -19580.037,E2 -19580.037} C_VEL
LIN {X 0,Y 242.294,Z 177.272,A -85,B 0,C 180,E1 -19582.097,E2 -19582.097} C_VEL
LIN {X 0,Y 239.465,Z 173.763,A -85,B 0,C 180,E1 -19583.144,E2 -19583.144} C_VEL
LIN {X 0,Y 238.568,Z 172.191,A -85,B 0,C 180,E1 -19583.509,E2 -19583.509} C_VEL
LIN {X 0,Y 236.226,Z 170.01,A -85,B 0,C 180,E1 -19584.392,E2 -19584.392} C_VEL
LIN {X 0,Y 235.091,Z 167.448,A -85,B 0,C 180,E1 -19585.049,E2 -19585.049} C_VEL
LIN {X 0,Y 234.956,Z 166.853,A -85,B 0,C 180,E1 -19585.577,E2 -19585.577} C_VEL
LIN {X 0,Y 234.97,Z 166.809,A -85,B 0,C 180,E1 -19590.157,E2 -19590.157} C_VEL
LIN {X 0,Y 234.995,Z 166.816,A -85,B 0,C 180,E1 -19593.794,E2 -19593.794} C_VEL
LIN {X 0,Y 235.013,Z 166.812,A -85,B 0,C 180,E1 -19598.97,E2 -19598.97} C_VEL
LIN {X 0,Y 235.098,Z 166.808,A -85,B 0,C 180,E1 -19603.06,E2 -19603.06} C_VEL
LIN {X 0,Y 235.144,Z 166.816,A -85,B 0,C 180,E1 -19607.924,E2 -19607.924} C_VEL
LIN {X 0,Y 235.313,Z 166.774,A -85,B 0,C 180,E1 -19611.412,E2 -19611.412} C_VEL
LIN {X 0,Y 235.352,Z 166.793,A -85,B 0,C 180,E1 -19613.14,E2 -19613.14} C_VEL
LIN {X 0,Y 235.593,Z 166.748,A -85,B 0,C 180,E1 -19618.291,E2 -19618.291} C_VEL
LIN {X 0,Y 235.583,Z 166.736,A -85,B 0,C 180,E1 -19621.71,E2 -19621.71} C_VEL
LIN {X 0,Y 235.352,Z 166.777,A -85,B 0,C 180,E1 -19626.86,E2 -19626.86} C_VEL
LIN {X 0,Y 235.215,Z 166.796,A -85,B 0,C 180,E1 -19630.328,E2 -19630.328} C_VEL
LIN {X 0,Y 235.075,Z 166.807,A -85,B 0,C 180,E1 -19635.609,E2 -19635.609} C_VEL
LIN {X 0,Y 234.97,Z 166.819,A -85,B 0,C 180,E1 -19639.209,E2 -19639.209} C_VEL
LIN {X 0,Y 234.909,Z 166.849,A -85,B 0,C 180,E1 -19642.888,E2 -19642.888} C_VEL
LIN {X 0,Y 234.926,Z 166.833,A -85,B 0,C 180,E1 -19646.663,E2 -19646.663} C_VEL
LIN {X 0,Y 234.899,Z 166.784,A -85,B 0,C 180,E1 -19650.573,E2 -19650.573} C_VEL
LIN {X 0,Y 234.941,Z 166.771,A -85,B 0,C 180,E1 -19653.114,E2 -19653.114} C_VEL
LIN {X 0,Y 234.955,Z 167.09,A -85,B 0,C 180,E1 -19654.927,E2 -19654.927} C_VEL
LIN {X 0,Y 235.253,Z 168.176,A -85,B 0,C 180,E1 -19655.337,E2 -19655.337} C_VEL
LIN {X 0,Y 236.661,Z 170.658,A -85,B 0,C 180,E1 -19655.964,E2 -19655.964} C_VEL
LIN {X 0,Y 238.946,Z 172.776,A -85,B 0,C 180,E1 -19656.819,E2 -19656.819} C_VEL
LIN {X 0,Y 241.02,Z 175.97,A -85,B 0,C 180,E1 -19657.628,E2 -19657.628} C_VEL
LIN {X 0,Y 242.677,Z 177.763,A -85,B 0,C 180,E1 -19658.218,E2 -19658.218} C_VEL
LIN {X 0,Y 245.362,Z 181.428,A -85,B 0,C 180,E1 -19659.177,E2 -19659.177} C_VEL
LIN {X 0,Y 252.257,Z 191.012,A -85,B 0,C 180,E1 -19661.473,E2 -19661.473} C_VEL
LIN {X 0,Y 257.418,Z 199.259,A -85,B 0,C 180,E1 -19663.092,E2 -19663.092} C_VEL
LIN {X 0,Y 265.508,Z 213.978,A -85,B 0,C 180,E1 -19665.483,E2 -19665.483} C_VEL
LIN {X 0,Y 272.304,Z 228.181,A -85,B 0,C 180,E1 -19667.378,E2 -19667.378} C_VEL
LIN {X 0,Y 274.866,Z 234.138,A -85,B 0,C 180,E1 -19668.075,E2 -19668.075} C_VEL
LIN {X 0,Y 270.307,Z 323.557,A -85,B 0,C 180,E1 -19670.31,E2 -19670.31} C_VEL
LIN {X 0,Y 268.975,Z 339.178,A -85,B 0,C 180,E1 -19670.863,E2 -19670.863} C_VEL
LIN {X 0,Y 266.932,Z 354.204,A -85,B 0,C 180,E1 -19671.657,E2 -19671.657} C_VEL
LIN {X 0,Y 264.787,Z 366.99,A -85,B 0,C 180,E1 -19672.583,E2 -19672.583} C_VEL
LIN {X 0,Y 262.011,Z 380.394,A -85,B 0,C 180,E1 -19673.835,E2 -19673.835} C_VEL
LIN {X 0,Y 258.594,Z 394.068,A -85,B 0,C 180,E1 -19675.435,E2 -19675.435} C_VEL
LIN {X 0,Y 254.633,Z 407.692,A -85,B 0,C 180,E1 -19677.438,E2 -19677.438} C_VEL
LIN {X 0,Y 250.714,Z 419.901,A -85,B 0,C 180,E1 -19679.697,E2 -19679.697} C_VEL
LIN {X 0,Y 247.022,Z 430.92,A -85,B 0,C 180,E1 -19682.238,E2 -19682.238} C_VEL
LIN {X 0,Y 243.655,Z 440.11,A -85,B 0,C 180,E1 -19684.821,E2 -19684.821} C_VEL
LIN {X 0,Y 240.605,Z 448.4,A -85,B 0,C 180,E1 -19687.683,E2 -19687.683} C_VEL
LIN {X 0,Y 237.549,Z 456.607,A -85,B 0,C 180,E1 -19691.216,E2 -19691.216} C_VEL
LIN {X 0,Y 235.679,Z 462.386,A -85,B 0,C 180,E1 -19694.432,E2 -19694.432} C_VEL
LIN {X 0,Y 234.152,Z 467.172,A -85,B 0,C 180,E1 -19697.872,E2 -19697.872} C_VEL
LIN {X 0,Y 233.202,Z 470.677,A -85,B 0,C 180,E1 -19701.333,E2 -19701.333} C_VEL
LIN {X 0,Y 232.725,Z 473.197,A -85,B 0,C 180,E1 -19705.248,E2 -19705.248} C_VEL
LIN {X 0,Y 232.685,Z 474.171,A -85,B 0,C 180,E1 -19708.269,E2 -19708.269} C_VEL
LIN {X 0,Y 232.72,Z 474.328,A -85,B 0,C 180,E1 -19710,E2 -19710} C_VEL
LIN {X 0,Y 232.689,Z 473.76,A -85,B 0,C 180,E1 -19713.463,E2 -19713.463} C_VEL
LIN {X 0,Y 232.916,Z 472.068,A -85,B 0,C 180,E1 -19716.932,E2 -19716.932} C_VEL
LIN {X 0,Y 233.605,Z 469.214,A -85,B 0,C 180,E1 -19720.4,E2 -19720.4} C_VEL
LIN {X 0,Y 234.741,Z 465.129,A -85,B 0,C 180,E1 -19723.858,E2 -19723.858} C_VEL
LIN {X 0,Y 236.566,Z 459.712,A -85,B 0,C 180,E1 -19727.283,E2 -19727.283} C_VEL
LIN {X 0,Y 239.024,Z 452.812,A -85,B 0,C 180,E1 -19730.661,E2 -19730.661} C_VEL
LIN {X 0,Y 242.219,Z 444.201,A -85,B 0,C 180,E1 -19733.967,E2 -19733.967} C_VEL
LIN {X 0,Y 245.682,Z 435.045,A -85,B 0,C 180,E1 -19736.779,E2 -19736.779} C_VEL
LIN {X 0,Y 248.269,Z 427.347,A -85,B 0,C 180,E1 -19738.766,E2 -19738.766} C_VEL
LIN {X 0,Y 251.909,Z 416.598,A -85,B 0,C 180,E1 -19741.073,E2 -19741.073} C_VEL
LIN {X 0,Y 255.598,Z 404.864,A -85,B 0,C 180,E1 -19743.127,E2 -19743.127} C_VEL
LIN {X 0,Y 259.214,Z 392.049,A -85,B 0,C 180,E1 -19744.943,E2 -19744.943} C_VEL
LIN {X 0,Y 262.45,Z 378.847,A -85,B 0,C 180,E1 -19746.444,E2 -19746.444} C_VEL
LIN {X 0,Y 265.14,Z 365.248,A -85,B 0,C 180,E1 -19747.685,E2 -19747.685} C_VEL
LIN {X 0,Y 267.535,Z 350.977,A -85,B 0,C 180,E1 -19748.662,E2 -19748.662} C_VEL
LIN {X 0,Y 269.481,Z 335.53,A -85,B 0,C 180,E1 -19749.411,E2 -19749.411} C_VEL
LIN {X 0,Y 270.671,Z 319.131,A -85,B 0,C 180,E1 -19749.928,E2 -19749.928} C_VEL
LIN {X 0,Y 275.026,Z 234.415,A -85,B 0,C 180,E1 -19752.028,E2 -19752.028} C_VEL
LIN {X 0,Y 269.257,Z 221.523,A -85,B 0,C 180,E1 -19753.61,E2 -19753.61} C_VEL
LIN {X 0,Y 263.002,Z 209.193,A -85,B 0,C 180,E1 -19755.392,E2 -19755.392} C_VEL
LIN {X 0,Y 256.004,Z 196.856,A -85,B 0,C 180,E1 -19757.506,E2 -19757.506} C_VEL
LIN {X 0,Y 251.35,Z 189.705,A -85,B 0,C 180,E1 -19758.983,E2 -19758.983} C_VEL
LIN {X 0,Y 245.228,Z 181.294,A -85,B 0,C 180,E1 -19761.041,E2 -19761.041} C_VEL
LIN {X 0,Y 242.54,Z 177.495,A -85,B 0,C 180,E1 -19762.013,E2 -19762.013} C_VEL
LIN {X 0,Y 239.584,Z 174.019,A -85,B 0,C 180,E1 -19763.099,E2 -19763.099} C_VEL
LIN {X 0,Y 238.583,Z 172.202,A -85,B 0,C 180,E1 -19763.511,E2 -19763.511} C_VEL
LIN {X 0,Y 236.28,Z 170.16,A -85,B 0,C 180,E1 -19764.378,E2 -19764.378} C_VEL
LIN {X 0,Y 235.011,Z 167.431,A -85,B 0,C 180,E1 -19765.083,E2 -19765.083} C_VEL
LIN {X 0,Y 234.926,Z 166.885,A -85,B 0,C 180,E1 -19765.573,E2 -19765.573} C_VEL
LIN {X 0,Y 234.899,Z 166.783,A -85,B 0,C 180,E1 -19769.427,E2 -19769.427} C_VEL
LIN {X 0,Y 234.942,Z 166.828,A -85,B 0,C 180,E1 -19773.82,E2 -19773.82} C_VEL
LIN {X 0,Y 234.938,Z 166.826,A -85,B 0,C 180,E1 -19778.963,E2 -19778.963} C_VEL
LIN {X 0,Y 235.056,Z 166.83,A -85,B 0,C 180,E1 -19783.093,E2 -19783.093} C_VEL
LIN {X 0,Y 235.1,Z 166.821,A -85,B 0,C 180,E1 -19787.921,E2 -19787.921} C_VEL
LIN {X 0,Y 235.314,Z 166.77,A -85,B 0,C 180,E1 -19791.412,E2 -19791.412} C_VEL
LIN {X 0,Y 235.353,Z 166.777,A -85,B 0,C 180,E1 -19793.14,E2 -19793.14} C_VEL
LIN {X 0,Y 235.353,Z 166.764,A -85,B 0,C 180,E1 -19797.128,E2 -19797.128} C_VEL
LIN {X 0,Y 234.825,Z 166.836,A -85,B 0,C 180,E1 -19798.559,E2 -19798.559} C_VEL
LIN {X 0,Y 233.257,Z 167.047,A -85,B 0,C 180,E1 -19799.964,E2 -19799.964} C_VEL
LIN {X 0,Y 229.377,Z 167.518,A -85,B 0,C 180,E1 -19802.792,E2 -19802.792} C_VEL
LIN {X 0,Y 228.256,Z 167.648,A -85,B 0,C 180,E1 -19804.272,E2 -19804.272} C_VEL
LIN {X 0,Y 228.16,Z 167.663,A -85,B 0,C 180,E1 -19804.775,E2 -19804.775} C_VEL
LIN {X 0,Y 228.305,Z 167.668,A -85,B 0,C 180,E1 -19807.073,E2 -19807.073} C_VEL
LIN {X 0,Y 228.151,Z 167.666,A -85,B 0,C 180,E1 -19810.651,E2 -19810.651} C_VEL
LIN {X 0,Y 228.066,Z 167.681,A -85,B 0,C 180,E1 -19814.272,E2 -19814.272} C_VEL
LIN {X 0,Y 228.004,Z 167.707,A -85,B 0,C 180,E1 -19817.953,E2 -19817.953} C_VEL
LIN {X 0,Y 227.918,Z 167.703,A -85,B 0,C 180,E1 -19822.321,E2 -19822.321} C_VEL
LIN {X 0,Y 227.944,Z 167.695,A -85,B 0,C 180,E1 -19826.602,E2 -19826.602} C_VEL
LIN {X 0,Y 227.91,Z 167.673,A -85,B 0,C 180,E1 -19830.296,E2 -19830.296} C_VEL
LIN {X 0,Y 227.908,Z 167.817,A -85,B 0,C 180,E1 -19831.876,E2 -19831.876} C_VEL
LIN {X 0,Y 228.128,Z 168.684,A -85,B 0,C 180,E1 -19832.428,E2 -19832.428} C_VEL
LIN {X 0,Y 229.574,Z 171.417,A -85,B 0,C 180,E1 -19833.195,E2 -19833.195} C_VEL
LIN {X 0,Y 232.003,Z 173.573,A -85,B 0,C 180,E1 -19834.215,E2 -19834.215} C_VEL
LIN {X 0,Y 234.076,Z 176.798,A -85,B 0,C 180,E1 -19835.122,E2 -19835.122} C_VEL
LIN {X 0,Y 236.037,Z 178.816,A -85,B 0,C 180,E1 -19835.895,E2 -19835.895} C_VEL
LIN {X 0,Y 238.662,Z 182.481,A -85,B 0,C 180,E1 -19836.935,E2 -19836.935} C_VEL
LIN {X 0,Y 241.002,Z 185.733,A -85,B 0,C 180,E1 -19837.823,E2 -19837.823} C_VEL
LIN {X 0,Y 247.459,Z 195.794,A -85,B 0,C 180,E1 -19840.151,E2 -19840.151} C_VEL
LIN {X 0,Y 254.403,Z 207.643,A -85,B 0,C 180,E1 -19842.456,E2 -19842.456} C_VEL
LIN {X 0,Y 261.667,Z 221.535,A -85,B 0,C 180,E1 -19844.697,E2 -19844.697} C_VEL
LIN {X 0,Y 268.399,Z 236.425,A -85,B 0,C 180,E1 -19846.668,E2 -19846.668} C_VEL
LIN {X 0,Y 269.564,Z 239.194,A -85,B 0,C 180,E1 -19846.999,E2 -19846.999} C_VEL
LIN {X 0,Y 264.589,Z 331.267,A -85,B 0,C 180,E1 -19849.338,E2 -19849.338} C_VEL
LIN {X 0,Y 263.073,Z 346.276,A -85,B 0,C 180,E1 -19849.934,E2 -19849.934} C_VEL
LIN {X 0,Y 260.881,Z 360.364,A -85,B 0,C 180,E1 -19850.722,E2 -19850.722} C_VEL
LIN {X 0,Y 257.941,Z 375.409,A -85,B 0,C 180,E1 -19851.88,E2 -19851.88} C_VEL
LIN {X 0,Y 254.871,Z 388.945,A -85,B 0,C 180,E1 -19853.269,E2 -19853.269} C_VEL
LIN {X 0,Y 251.148,Z 402.437,A -85,B 0,C 180,E1 -19854.994,E2 -19854.994} C_VEL
LIN {X 0,Y 247.082,Z 415.27,A -85,B 0,C 180,E1 -19857.044,E2 -19857.044} C_VEL
LIN {X 0,Y 243.407,Z 426.013,A -85,B 0,C 180,E1 -19859.169,E2 -19859.169} C_VEL
LIN {X 0,Y 239.932,Z 435.69,A -85,B 0,C 180,E1 -19861.491,E2 -19861.491} C_VEL
LIN {X 0,Y 236.231,Z 445.679,A -85,B 0,C 180,E1 -19864.444,E2 -19864.444} C_VEL
LIN {X 0,Y 233.054,Z 453.792,A -85,B 0,C 180,E1 -19867.388,E2 -19867.388} C_VEL
LIN {X 0,Y 229.973,Z 461.906,A -85,B 0,C 180,E1 -19871.134,E2 -19871.134} C_VEL
LIN {X 0,Y 227.954,Z 468.011,A -85,B 0,C 180,E1 -19874.807,E2 -19874.807} C_VEL
LIN {X 0,Y 226.814,Z 471.485,A -85,B 0,C 180,E1 -19877.473,E2 -19877.473} C_VEL
LIN {X 0,Y 225.98,Z 474.994,A -85,B 0,C 180,E1 -19881.054,E2 -19881.054} C_VEL
LIN {X 0,Y 225.589,Z 477.301,A -85,B 0,C 180,E1 -19884.637,E2 -19884.637} C_VEL
LIN {X 0,Y 225.544,Z 478.46,A -85,B 0,C 180,E1 -19888.214,E2 -19888.214} C_VEL
LIN {X 0,Y 225.631,Z 478.613,A -85,B 0,C 180,E1 -19890,E2 -19890} C_VEL
LIN {X 0,Y 225.521,Z 478.008,A -85,B 0,C 180,E1 -19893.573,E2 -19893.573} C_VEL
LIN {X 0,Y 225.734,Z 476.262,A -85,B 0,C 180,E1 -19897.154,E2 -19897.154} C_VEL
LIN {X 0,Y 226.33,Z 473.348,A -85,B 0,C 180,E1 -19900.738,E2 -19900.738} C_VEL
LIN {X 0,Y 227.552,Z 469.2,A -85,B 0,C 180,E1 -19904.305,E2 -19904.305} C_VEL
LIN {X 0,Y 229.325,Z 463.705,A -85,B 0,C 180,E1 -19907.846,E2 -19907.846} C_VEL
LIN {X 0,Y 231.892,Z 456.715,A -85,B 0,C 180,E1 -19911.327,E2 -19911.327} C_VEL
LIN {X 0,Y 235.171,Z 448.018,A -85,B 0,C 180,E1 -19914.733,E2 -19914.733} C_VEL
LIN {X 0,Y 238.225,Z 440.223,A -85,B 0,C 180,E1 -19917.211,E2 -19917.211} C_VEL
LIN {X 0,Y 240.924,Z 432.651,A -85,B 0,C 180,E1 -19919.249,E2 -19919.249} C_VEL
LIN {X 0,Y 244.736,Z 422.129,A -85,B 0,C 180,E1 -19921.606,E2 -19921.606} C_VEL
LIN {X 0,Y 248.492,Z 410.686,A -85,B 0,C 180,E1 -19923.714,E2 -19923.714} C_VEL
LIN {X 0,Y 252.297,Z 398.243,A -85,B 0,C 180,E1 -19925.556,E2 -19925.556} C_VEL
LIN {X 0,Y 255.857,Z 384.604,A -85,B 0,C 180,E1 -19927.179,E2 -19927.179} C_VEL
LIN {X 0,Y 258.862,Z 370.465,A -85,B 0,C 180,E1 -19928.517,E2 -19928.517} C_VEL
LIN {X 0,Y 261.547,Z 355.896,A -85,B 0,C 180,E1 -19929.532,E2 -19929.532} C_VEL
LIN {X 0,Y 263.557,Z 340.919,A -85,B 0,C 180,E1 -19930.289,E2 -19930.289} C_VEL
LIN {X 0,Y 264.85,Z 325.456,A -85,B 0,C 180,E1 -19930.802,E2 -19930.802} C_VEL
LIN {X 0,Y 269.474,Z 239.745,A -85,B 0,C 180,E1 -19932.943,E2 -19932.943} C_VEL
LIN {X 0,Y 268.557,Z 236.934,A -85,B 0,C 180,E1 -19933.226,E2 -19933.226} C_VEL
LIN {X 0,Y 261.412,Z 221.049,A -85,B 0,C 180,E1 -19935.315,E2 -19935.315} C_VEL
LIN {X 0,Y 253.623,Z 206.261,A -85,B 0,C 180,E1 -19937.723,E2 -19937.723} C_VEL
LIN {X 0,Y 245.542,Z 192.688,A -85,B 0,C 180,E1 -19940.44,E2 -19940.44} C_VEL
LIN {X 0,Y 238.977,Z 182.79,A -85,B 0,C 180,E1 -19942.858,E2 -19942.858} C_VEL
LIN {X 0,Y 236.193,Z 179.133,A -85,B 0,C 180,E1 -19943.94,E2 -19943.94} C_VEL
LIN {X 0,Y 235.112,Z 177.824,A -85,B 0,C 180,E1 -19944.369,E2 -19944.369} C_VEL
LIN {X 0,Y 232.676,Z 174.788,A -85,B 0,C 180,E1 -19945.373,E2 -19945.373} C_VEL
LIN {X 0,Y 231.607,Z 173.072,A -85,B 0,C 180,E1 -19945.849,E2 -19945.849} C_VEL
LIN {X 0,Y 229.286,Z 171.05,A -85,B 0,C 180,E1 -19946.824,E2 -19946.824} C_VEL
LIN {X 0,Y 228.031,Z 168.267,A -85,B 0,C 180,E1 -19947.622,E2 -19947.622} C_VEL
LIN {X 0,Y 227.873,Z 167.7,A -85,B 0,C 180,E1 -19948.379,E2 -19948.379} C_VEL
LIN {X 0,Y 227.888,Z 167.71,A -85,B 0,C 180,E1 -19952.446,E2 -19952.446} C_VEL
LIN {X 0,Y 227.916,Z 167.721,A -85,B 0,C 180,E1 -19956.368,E2 -19956.368} C_VEL
LIN {X 0,Y 227.944,Z 167.698,A -85,B 0,C 180,E1 -19960.175,E2 -19960.175} C_VEL
LIN {X 0,Y 228.059,Z 167.677,A -85,B 0,C 180,E1 -19963.898,E2 -19963.898} C_VEL
LIN {X 0,Y 228.092,Z 167.699,A -85,B 0,C 180,E1 -19967.545,E2 -19967.545} C_VEL
LIN {X 0,Y 228.254,Z 167.651,A -85,B 0,C 180,E1 -19971.144,E2 -19971.144} C_VEL
LIN {X 0,Y 228.304,Z 167.668,A -85,B 0,C 180,E1 -19972.927,E2 -19972.927} C_VEL
LIN {X 0,Y 228.552,Z 167.623,A -85,B 0,C 180,E1 -19978.238,E2 -19978.238} C_VEL
LIN {X 0,Y 228.541,Z 167.612,A -85,B 0,C 180,E1 -19981.762,E2 -19981.762} C_VEL
LIN {X 0,Y 228.304,Z 167.651,A -85,B 0,C 180,E1 -19987.073,E2 -19987.073} C_VEL
LIN {X 0,Y 228.146,Z 167.681,A -85,B 0,C 180,E1 -19990.651,E2 -19990.651} C_VEL
LIN {X 0,Y 228.042,Z 167.677,A -85,B 0,C 180,E1 -19994.274,E2 -19994.274} C_VEL
LIN {X 0,Y 227.931,Z 167.711,A -85,B 0,C 180,E1 -19997.959,E2 -19997.959} C_VEL
LIN {X 0,Y 227.89,Z 167.72,A -85,B 0,C 180,E1 -20002.304,E2 -20002.304} C_VEL
LIN {X 0,Y 227.904,Z 167.707,A -85,B 0,C 180,E1 -20006.583,E2 -20006.583} C_VEL
LIN {X 0,Y 227.873,Z 167.662,A -85,B 0,C 180,E1 -20010.28,E2 -20010.28} C_VEL
LIN {X 0,Y 227.936,Z 167.985,A -85,B 0,C 180,E1 -20012.328,E2 -20012.328} C_VEL
LIN {X 0,Y 228.225,Z 169.03,A -85,B 0,C 180,E1 -20012.806,E2 -20012.806} C_VEL
LIN {X 0,Y 229.822,Z 171.751,A -85,B 0,C 180,E1 -20013.595,E2 -20013.595} C_VEL
LIN {X 0,Y 231.973,Z 173.519,A -85,B 0,C 180,E1 -20014.484,E2 -20014.484} C_VEL
LIN {X 0,Y 234.025,Z 176.791,A -85,B 0,C 180,E1 -20015.381,E2 -20015.381} C_VEL
LIN {X 0,Y 236.113,Z 178.984,A -85,B 0,C 180,E1 -20016.202,E2 -20016.202} C_VEL
LIN {X 0,Y 238.535,Z 182.347,A -85,B 0,C 180,E1 -20017.157,E2 -20017.157} C_VEL
LIN {X 0,Y 239.835,Z 184.027,A -85,B 0,C 180,E1 -20017.647,E2 -20017.647} C_VEL
LIN {X 0,Y 243.466,Z 188.97,A -85,B 0,C 180,E1 -20018.973,E2 -20018.973} C_VEL
LIN {X 0,Y 249.488,Z 197.605,A -85,B 0,C 180,E1 -20021.03,E2 -20021.03} C_VEL
LIN {X 0,Y 254.896,Z 206.591,A -85,B 0,C 180,E1 -20022.78,E2 -20022.78} C_VEL
LIN {X 0,Y 262.69,Z 221.359,A -85,B 0,C 180,E1 -20025.153,E2 -20025.153} C_VEL
LIN {X 0,Y 269.07,Z 235.449,A -85,B 0,C 180,E1 -20027,E2 -20027} C_VEL
LIN {X 0,Y 269.494,Z 236.43,A -85,B 0,C 180,E1 -20027.119,E2 -20027.119} C_VEL
LIN {X 0,Y 265.308,Z 316.862,A -85,B 0,C 180,E1 -20029.158,E2 -20029.158} C_VEL
LIN {X 0,Y 264.038,Z 334.117,A -85,B 0,C 180,E1 -20029.674,E2 -20029.674} C_VEL
LIN {X 0,Y 262.181,Z 349.302,A -85,B 0,C 180,E1 -20030.396,E2 -20030.396} C_VEL
LIN {X 0,Y 259.683,Z 364.012,A -85,B 0,C 180,E1 -20031.38,E2 -20031.38} C_VEL
LIN {X 0,Y 256.812,Z 378.2,A -85,B 0,C 180,E1 -20032.666,E2 -20032.666} C_VEL
LIN {X 0,Y 253.561,Z 391.289,A -85,B 0,C 180,E1 -20034.16,E2 -20034.16} C_VEL
LIN {X 0,Y 249.763,Z 404.257,A -85,B 0,C 180,E1 -20035.996,E2 -20035.996} C_VEL
LIN {X 0,Y 245.944,Z 416.098,A -85,B 0,C 180,E1 -20038.086,E2 -20038.086} C_VEL
LIN {X 0,Y 242.131,Z 426.936,A -85,B 0,C 180,E1 -20040.433,E2 -20040.433} C_VEL
LIN {X 0,Y 238.319,Z 437.478,A -85,B 0,C 180,E1 -20043.274,E2 -20043.274} C_VEL
LIN {X 0,Y 234.877,Z 446.243,A -85,B 0,C 180,E1 -20046.175,E2 -20046.175} C_VEL
LIN {X 0,Y 232.388,Z 452.575,A -85,B 0,C 180,E1 -20048.721,E2 -20048.721} C_VEL
LIN {X 0,Y 229.782,Z 459.541,A -85,B 0,C 180,E1 -20052.19,E2 -20052.19} C_VEL
LIN {X 0,Y 227.846,Z 465.015,A -85,B 0,C 180,E1 -20055.714,E2 -20055.714} C_VEL
LIN {X 0,Y 226.615,Z 469.145,A -85,B 0,C 180,E1 -20059.276,E2 -20059.276} C_VEL
LIN {X 0,Y 225.886,Z 472.046,A -85,B 0,C 180,E1 -20062.851,E2 -20062.851} C_VEL
LIN {X 0,Y 225.604,Z 473.788,A -85,B 0,C 180,E1 -20066.428,E2 -20066.428} C_VEL
LIN {X 0,Y 225.636,Z 474.394,A -85,B 0,C 180,E1 -20070,E2 -20070} C_VEL
LIN {X 0,Y 225.602,Z 473.826,A -85,B 0,C 180,E1 -20073.572,E2 -20073.572} C_VEL
LIN {X 0,Y 225.841,Z 472.135,A -85,B 0,C 180,E1 -20077.151,E2 -20077.151} C_VEL
LIN {X 0,Y 226.585,Z 469.28,A -85,B 0,C 180,E1 -20080.726,E2 -20080.726} C_VEL
LIN {X 0,Y 227.821,Z 465.194,A -85,B 0,C 180,E1 -20084.288,E2 -20084.288} C_VEL
LIN {X 0,Y 229.756,Z 459.778,A -85,B 0,C 180,E1 -20087.812,E2 -20087.812} C_VEL
LIN {X 0,Y 232.353,Z 452.877,A -85,B 0,C 180,E1 -20091.283,E2 -20091.283} C_VEL
LIN {X 0,Y 235.688,Z 444.265,A -85,B 0,C 180,E1 -20094.675,E2 -20094.675} C_VEL
LIN {X 0,Y 239.312,Z 435.109,A -85,B 0,C 180,E1 -20097.551,E2 -20097.551} C_VEL
LIN {X 0,Y 242.025,Z 427.411,A -85,B 0,C 180,E1 -20099.581,E2 -20099.581} C_VEL
LIN {X 0,Y 245.84,Z 416.661,A -85,B 0,C 180,E1 -20101.93,E2 -20101.93} C_VEL
LIN {X 0,Y 249.68,Z 404.926,A -85,B 0,C 180,E1 -20104.017,E2 -20104.017} C_VEL
LIN {X 0,Y 253.411,Z 392.111,A -85,B 0,C 180,E1 -20105.865,E2 -20105.865} C_VEL
LIN {X 0,Y 256.884,Z 378.356,A -85,B 0,C 180,E1 -20107.443,E2 -20107.443} C_VEL
LIN {X 0,Y 259.776,Z 364.178,A -85,B 0,C 180,E1 -20108.728,E2 -20108.728} C_VEL
LIN {X 0,Y 262.249,Z 349.51,A -85,B 0,C 180,E1 -20109.717,E2 -20109.717} C_VEL
LIN {X 0,Y 264.15,Z 334.441,A -85,B 0,C 180,E1 -20110.431,E2 -20110.431} C_VEL
LIN {X 0,Y 265.389,Z 317.385,A -85,B 0,C 180,E1 -20110.952,E2 -20110.952} C_VEL
LIN {X 0,Y 269.656,Z 236.738,A -85,B 0,C 180,E1 -20112.984,E2 -20112.984} C_VEL
LIN {X 0,Y 264.604,Z 225.328,A -85,B 0,C 180,E1 -20114.437,E2 -20114.437} C_VEL
LIN {X 0,Y 258.537,Z 213.207,A -85,B 0,C 180,E1 -20116.248,E2 -20116.248} C_VEL
LIN {X 0,Y 251.61,Z 200.885,A -85,B 0,C 180,E1 -20118.441,E2 -20118.441} C_VEL
LIN {X 0,Y 246.873,Z 193.767,A -85,B 0,C 180,E1 -20120.013,E2 -20120.013} C_VEL
LIN {X 0,Y 241.828,Z 186.705,A -85,B 0,C 180,E1 -20121.794,E2 -20121.794} C_VEL
LIN {X 0,Y 238.628,Z 182.422,A -85,B 0,C 180,E1 -20122.992,E2 -20122.992} C_VEL
LIN {X 0,Y 236.028,Z 178.866,A -85,B 0,C 180,E1 -20124.019,E2 -20124.019} C_VEL
LIN {X 0,Y 232.804,Z 175.1,A -85,B 0,C 180,E1 -20125.329,E2 -20125.329} C_VEL
LIN {X 0,Y 231.64,Z 173.121,A -85,B 0,C 180,E1 -20125.855,E2 -20125.855} C_VEL
LIN {X 0,Y 229.208,Z 170.929,A -85,B 0,C 180,E1 -20126.886,E2 -20126.886} C_VEL
LIN {X 0,Y 228.024,Z 168.393,A -85,B 0,C 180,E1 -20127.621,E2 -20127.621} C_VEL
LIN {X 0,Y 227.857,Z 167.728,A -85,B 0,C 180,E1 -20128.376,E2 -20128.376} C_VEL
LIN {X 0,Y 227.846,Z 167.73,A -85,B 0,C 180,E1 -20132.44,E2 -20132.44} C_VEL
LIN {X 0,Y 227.858,Z 167.713,A -85,B 0,C 180,E1 -20136.361,E2 -20136.361} C_VEL
LIN {X 0,Y 227.892,Z 167.697,A -85,B 0,C 180,E1 -20140.17,E2 -20140.17} C_VEL
LIN {X 0,Y 228.019,Z 167.692,A -85,B 0,C 180,E1 -20143.895,E2 -20143.895} C_VEL
LIN {X 0,Y 228.144,Z 167.683,A -85,B 0,C 180,E1 -20149.349,E2 -20149.349} C_VEL
LIN {X 0,Y 228.305,Z 167.651,A -85,B 0,C 180,E1 -20152.927,E2 -20152.927} C_VEL
LIN {X 0,Y 228.541,Z 167.612,A -85,B 0,C 180,E1 -20158.238,E2 -20158.238} C_VEL
LIN {X 0,Y 228.55,Z 167.624,A -85,B 0,C 180,E1 -20161.762,E2 -20161.762} C_VEL
LIN {X 0,Y 228.16,Z 167.663,A -85,B 0,C 180,E1 -20164.775,E2 -20164.775} C_VEL
LIN {X 0,Y 227.466,Z 167.771,A -85,B 0,C 180,E1 -20166.251,E2 -20166.251} C_VEL
LIN {X 0,Y 224.568,Z 168.115,A -85,B 0,C 180,E1 -20168.657,E2 -20168.657} C_VEL
LIN {X 0,Y 222.125,Z 168.417,A -85,B 0,C 180,E1 -20170.621,E2 -20170.621} C_VEL
LIN {X 0,Y 221.096,Z 168.566,A -85,B 0,C 180,E1 -20172.147,E2 -20172.147} C_VEL
LIN {X 0,Y 221.022,Z 168.575,A -85,B 0,C 180,E1 -20172.664,E2 -20172.664} C_VEL
LIN {X 0,Y 220.986,Z 168.571,A -85,B 0,C 180,E1 -20177.428,E2 -20177.428} C_VEL
LIN {X 0,Y 220.886,Z 168.582,A -85,B 0,C 180,E1 -20182.675,E2 -20182.675} C_VEL
LIN {X 0,Y 220.887,Z 168.577,A -85,B 0,C 180,E1 -20187.015,E2 -20187.015} C_VEL
LIN {X 0,Y 220.878,Z 168.838,A -85,B 0,C 180,E1 -20189.027,E2 -20189.027} C_VEL
LIN {X 0,Y 221.171,Z 169.829,A -85,B 0,C 180,E1 -20189.572,E2 -20189.572} C_VEL
LIN {X 0,Y 222.599,Z 172.399,A -85,B 0,C 180,E1 -20190.407,E2 -20190.407} C_VEL
LIN {X 0,Y 225.212,Z 174.501,A -85,B 0,C 180,E1 -20191.645,E2 -20191.645} C_VEL
LIN {X 0,Y 227.136,Z 177.655,A -85,B 0,C 180,E1 -20192.604,E2 -20192.604} C_VEL
LIN {X 0,Y 229.339,Z 179.856,A -85,B 0,C 180,E1 -20193.575,E2 -20193.575} C_VEL
LIN {X 0,Y 231.995,Z 183.492,A -85,B 0,C 180,E1 -20194.743,E2 -20194.743} C_VEL
LIN {X 0,Y 233.434,Z 185.237,A -85,B 0,C 180,E1 -20195.339,E2 -20195.339} C_VEL
LIN {X 0,Y 237.5,Z 190.829,A -85,B 0,C 180,E1 -20196.974,E2 -20196.974} C_VEL
LIN {X 0,Y 243.704,Z 200.688,A -85,B 0,C 180,E1 -20199.318,E2 -20199.318} C_VEL
LIN {X 0,Y 250.45,Z 212.384,A -85,B 0,C 180,E1 -20201.66,E2 -20201.66} C_VEL
LIN {X 0,Y 257.361,Z 225.829,A -85,B 0,C 180,E1 -20203.891,E2 -20203.891} C_VEL
LIN {X 0,Y 263.792,Z 240.324,A -85,B 0,C 180,E1 -20205.863,E2 -20205.863} C_VEL
LIN {X 0,Y 264.285,Z 241.935,A -85,B 0,C 180,E1 -20206.026,E2 -20206.026} C_VEL
LIN {X 0,Y 259.243,Z 331.219,A -85,B 0,C 180,E1 -20208.315,E2 -20208.315} C_VEL
LIN {X 0,Y 257.688,Z 346.221,A -85,B 0,C 180,E1 -20208.92,E2 -20208.92} C_VEL
LIN {X 0,Y 255.427,Z 360.305,A -85,B 0,C 180,E1 -20209.714,E2 -20209.714} C_VEL
LIN {X 0,Y 252.69,Z 373.856,A -85,B 0,C 180,E1 -20210.747,E2 -20210.747} C_VEL
LIN {X 0,Y 249.267,Z 388.632,A -85,B 0,C 180,E1 -20212.261,E2 -20212.261} C_VEL
LIN {X 0,Y 245.34,Z 402.374,A -85,B 0,C 180,E1 -20214.038,E2 -20214.038} C_VEL
LIN {X 0,Y 241.145,Z 415.206,A -85,B 0,C 180,E1 -20216.125,E2 -20216.125} C_VEL
LIN {X 0,Y 237.299,Z 425.949,A -85,B 0,C 180,E1 -20218.285,E2 -20218.285} C_VEL
LIN {X 0,Y 233.454,Z 436.19,A -85,B 0,C 180,E1 -20220.812,E2 -20220.812} C_VEL
LIN {X 0,Y 229.811,Z 445.614,A -85,B 0,C 180,E1 -20223.677,E2 -20223.677} C_VEL
LIN {X 0,Y 226.454,Z 453.726,A -85,B 0,C 180,E1 -20226.69,E2 -20226.69} C_VEL
LIN {X 0,Y 223.772,Z 460.436,A -85,B 0,C 180,E1 -20229.789,E2 -20229.789} C_VEL
LIN {X 0,Y 221.491,Z 466.63,A -85,B 0,C 180,E1 -20233.407,E2 -20233.407} C_VEL
LIN {X 0,Y 219.839,Z 471.419,A -85,B 0,C 180,E1 -20237.069,E2 -20237.069} C_VEL
LIN {X 0,Y 218.941,Z 474.928,A -85,B 0,C 180,E1 -20240.764,E2 -20240.764} C_VEL
LIN {X 0,Y 218.5,Z 477.235,A -85,B 0,C 180,E1 -20244.463,E2 -20244.463} C_VEL
LIN {X 0,Y 218.447,Z 478.394,A -85,B 0,C 180,E1 -20248.156,E2 -20248.156} C_VEL
LIN {X 0,Y 218.529,Z 478.547,A -85,B 0,C 180,E1 -20250,E2 -20250} C_VEL
LIN {X 0,Y 218.428,Z 477.828,A -85,B 0,C 180,E1 -20254.105,E2 -20254.105} C_VEL
LIN {X 0,Y 218.653,Z 476.195,A -85,B 0,C 180,E1 -20257.387,E2 -20257.387} C_VEL
LIN {X 0,Y 219.3,Z 473.281,A -85,B 0,C 180,E1 -20261.086,E2 -20261.086} C_VEL
LIN {X 0,Y 220.613,Z 469.132,A -85,B 0,C 180,E1 -20264.765,E2 -20264.765} C_VEL
LIN {X 0,Y 222.51,Z 463.636,A -85,B 0,C 180,E1 -20268.412,E2 -20268.412} C_VEL
LIN {X 0,Y 225.226,Z 456.646,A -85,B 0,C 180,E1 -20271.99,E2 -20271.99} C_VEL
LIN {X 0,Y 228.712,Z 447.949,A -85,B 0,C 180,E1 -20275.48,E2 -20275.48} C_VEL
LIN {X 0,Y 232.219,Z 439.155,A -85,B 0,C 180,E1 -20278.32,E2 -20278.32} C_VEL
LIN {X 0,Y 236.002,Z 429.315,A -85,B 0,C 180,E1 -20280.91,E2 -20280.91} C_VEL
LIN {X 0,Y 240.423,Z 417.125,A -85,B 0,C 180,E1 -20283.487,E2 -20283.487} C_VEL
LIN {X 0,Y 244.515,Z 404.69,A -85,B 0,C 180,E1 -20285.594,E2 -20285.594} C_VEL
LIN {X 0,Y 248.259,Z 392.196,A -85,B 0,C 180,E1 -20287.283,E2 -20287.283} C_VEL
LIN {X 0,Y 251.445,Z 379.23,A -85,B 0,C 180,E1 -20288.711,E2 -20288.711} C_VEL
LIN {X 0,Y 254.252,Z 365.878,A -85,B 0,C 180,E1 -20289.862,E2 -20289.862} C_VEL
LIN {X 0,Y 256.833,Z 351.261,A -85,B 0,C 180,E1 -20290.792,E2 -20290.792} C_VEL
LIN {X 0,Y 258.673,Z 336.334,A -85,B 0,C 180,E1 -20291.472,E2 -20291.472} C_VEL
LIN {X 0,Y 260.032,Z 316.437,A -85,B 0,C 180,E1 -20292.05,E2 -20292.05} C_VEL
LIN {X 0,Y 264.187,Z 241.491,A -85,B 0,C 180,E1 -20293.952,E2 -20293.952} C_VEL
LIN {X 0,Y 258.436,Z 228.306,A -85,B 0,C 180,E1 -20295.701,E2 -20295.701} C_VEL
LIN {X 0,Y 251.935,Z 215.233,A -85,B 0,C 180,E1 -20297.772,E2 -20297.772} C_VEL
LIN {X 0,Y 246.304,Z 205.251,A -85,B 0,C 180,E1 -20299.67,E2 -20299.67} C_VEL
LIN {X 0,Y 241.165,Z 196.611,A -85,B 0,C 180,E1 -20301.528,E2 -20301.528} C_VEL
LIN {X 0,Y 235.789,Z 188.413,A -85,B 0,C 180,E1 -20303.606,E2 -20303.606} C_VEL
LIN {X 0,Y 232.275,Z 183.748,A -85,B 0,C 180,E1 -20305.041,E2 -20305.041} C_VEL
LIN {X 0,Y 229.744,Z 180.486,A -85,B 0,C 180,E1 -20306.129,E2 -20306.129} C_VEL
LIN {X 0,Y 228.804,Z 179.17,A -85,B 0,C 180,E1 -20306.554,E2 -20306.554} C_VEL
LIN {X 0,Y 226.22,Z 176.438,A -85,B 0,C 180,E1 -20307.713,E2 -20307.713} C_VEL
LIN {X 0,Y 225.028,Z 174.214,A -85,B 0,C 180,E1 -20308.326,E2 -20308.326} C_VEL
LIN {X 0,Y 222.502,Z 172.295,A -85,B 0,C 180,E1 -20309.512,E2 -20309.512} C_VEL
LIN {X 0,Y 221.025,Z 169.343,A -85,B 0,C 180,E1 -20310.472,E2 -20310.472} C_VEL
LIN {X 0,Y 220.839,Z 168.649,A -85,B 0,C 180,E1 -20311.227,E2 -20311.227} C_VEL
LIN {X 0,Y 220.896,Z 168.572,A -85,B 0,C 180,E1 -20313.55,E2 -20313.55} C_VEL
LIN {X 0,Y 220.88,Z 168.579,A -85,B 0,C 180,E1 -20317.554,E2 -20317.554} C_VEL
LIN {X 0,Y 220.986,Z 168.571,A -85,B 0,C 180,E1 -20322.571,E2 -20322.571} C_VEL
LIN {X 0,Y 221.025,Z 168.579,A -85,B 0,C 180,E1 -20327.14,E2 -20327.14} C_VEL
LIN {X 0,Y 221.195,Z 168.528,A -85,B 0,C 180,E1 -20330.859,E2 -20330.859} C_VEL
LIN {X 0,Y 221.124,Z 168.547,A -85,B 0,C 180,E1 -20334.529,E2 -20334.529} C_VEL
LIN {X 0,Y 221.509,Z 168.498,A -85,B 0,C 180,E1 -20338.182,E2 -20338.182} C_VEL
LIN {X 0,Y 221.474,Z 168.491,A -85,B 0,C 180,E1 -20341.819,E2 -20341.819} C_VEL
LIN {X 0,Y 221.242,Z 168.528,A -85,B 0,C 180,E1 -20347.3,E2 -20347.3} C_VEL
LIN {X 0,Y 221.081,Z 168.567,A -85,B 0,C 180,E1 -20350.996,E2 -20350.996} C_VEL
LIN {X 0,Y 220.979,Z 168.575,A -85,B 0,C 180,E1 -20356.633,E2 -20356.633} C_VEL
LIN {X 0,Y 220.852,Z 168.574,A -85,B 0,C 180,E1 -20360.49,E2 -20360.49} C_VEL
LIN {X 0,Y 220.797,Z 168.586,A -85,B 0,C 180,E1 -20364.443,E2 -20364.443} C_VEL
LIN {X 0,Y 220.8,Z 168.598,A -85,B 0,C 180,E1 -20368.519,E2 -20368.519} C_VEL
LIN {X 0,Y 220.867,Z 168.884,A -85,B 0,C 180,E1 -20369.421,E2 -20369.421} C_VEL
LIN {X 0,Y 221.249,Z 170.15,A -85,B 0,C 180,E1 -20369.955,E2 -20369.955} C_VEL
LIN {X 0,Y 222.832,Z 172.695,A -85,B 0,C 180,E1 -20370.832,E2 -20370.832} C_VEL
LIN {X 0,Y 225.252,Z 174.649,A -85,B 0,C 180,E1 -20371.968,E2 -20371.968} C_VEL
LIN {X 0,Y 227.311,Z 177.92,A -85,B 0,C 180,E1 -20372.979,E2 -20372.979} C_VEL
LIN {X 0,Y 229.354,Z 179.914,A -85,B 0,C 180,E1 -20373.87,E2 -20373.87} C_VEL
LIN {X 0,Y 231.848,Z 183.414,A -85,B 0,C 180,E1 -20374.967,E2 -20374.967} C_VEL
LIN {X 0,Y 233.37,Z 185.189,A -85,B 0,C 180,E1 -20375.592,E2 -20375.592} C_VEL
LIN {X 0,Y 237.33,Z 190.601,A -85,B 0,C 180,E1 -20377.178,E2 -20377.178} C_VEL
LIN {X 0,Y 242.827,Z 198.249,A -85,B 0,C 180,E1 -20379.214,E2 -20379.214} C_VEL
LIN {X 0,Y 247.792,Z 205.853,A -85,B 0,C 180,E1 -20380.936,E2 -20380.936} C_VEL
LIN {X 0,Y 254.342,Z 217.742,A -85,B 0,C 180,E1 -20383.098,E2 -20383.098} C_VEL
LIN {X 0,Y 260.333,Z 229.904,A -85,B 0,C 180,E1 -20384.962,E2 -20384.962} C_VEL
LIN {X 0,Y 264.247,Z 238.868,A -85,B 0,C 180,E1 -20386.14,E2 -20386.14} C_VEL
LIN {X 0,Y 259.142,Z 329.631,A -85,B 0,C 180,E1 -20388.49,E2 -20388.49} C_VEL
LIN {X 0,Y 257.304,Z 345.57,A -85,B 0,C 180,E1 -20389.169,E2 -20389.169} C_VEL
LIN {X 0,Y 254.827,Z 360.705,A -85,B 0,C 180,E1 -20390.117,E2 -20390.117} C_VEL
LIN {X 0,Y 251.846,Z 375.414,A -85,B 0,C 180,E1 -20391.386,E2 -20391.386} C_VEL
LIN {X 0,Y 248.622,Z 388.506,A -85,B 0,C 180,E1 -20392.827,E2 -20392.827} C_VEL
LIN {X 0,Y 244.689,Z 401.984,A -85,B 0,C 180,E1 -20394.688,E2 -20394.688} C_VEL
LIN {X 0,Y 241.002,Z 413.178,A -85,B 0,C 180,E1 -20396.604,E2 -20396.604} C_VEL
LIN {X 0,Y 237.169,Z 423.599,A -85,B 0,C 180,E1 -20398.763,E2 -20398.763} C_VEL
LIN {X 0,Y 233.63,Z 433.264,A -85,B 0,C 180,E1 -20401.229,E2 -20401.229} C_VEL
LIN {X 0,Y 229.76,Z 442.743,A -85,B 0,C 180,E1 -20404.158,E2 -20404.158} C_VEL
LIN {X 0,Y 226.168,Z 451.639,A -85,B 0,C 180,E1 -20407.625,E2 -20407.625} C_VEL
LIN {X 0,Y 223.49,Z 458.196,A -85,B 0,C 180,E1 -20410.835,E2 -20410.835} C_VEL
LIN {X 0,Y 221.46,Z 463.845,A -85,B 0,C 180,E1 -20414.351,E2 -20414.351} C_VEL
LIN {X 0,Y 220.182,Z 467.307,A -85,B 0,C 180,E1 -20417.089,E2 -20417.089} C_VEL
LIN {X 0,Y 219.13,Z 470.811,A -85,B 0,C 180,E1 -20420.772,E2 -20420.772} C_VEL
LIN {X 0,Y 218.602,Z 473.126,A -85,B 0,C 180,E1 -20424.465,E2 -20424.465} C_VEL
LIN {X 0,Y 218.489,Z 474.304,A -85,B 0,C 180,E1 -20428.157,E2 -20428.157} C_VEL
LIN {X 0,Y 218.536,Z 474.461,A -85,B 0,C 180,E1 -20430,E2 -20430} C_VEL
LIN {X 0,Y 218.502,Z 473.893,A -85,B 0,C 180,E1 -20433.688,E2 -20433.688} C_VEL
LIN {X 0,Y 218.791,Z 472.201,A -85,B 0,C 180,E1 -20437.382,E2 -20437.382} C_VEL
LIN {X 0,Y 219.584,Z 469.346,A -85,B 0,C 180,E1 -20441.072,E2 -20441.072} C_VEL
LIN {X 0,Y 220.921,Z 465.26,A -85,B 0,C 180,E1 -20444.744,E2 -20444.744} C_VEL
LIN {X 0,Y 222.957,Z 459.843,A -85,B 0,C 180,E1 -20448.374,E2 -20448.374} C_VEL
LIN {X 0,Y 225.7,Z 452.943,A -85,B 0,C 180,E1 -20451.942,E2 -20451.942} C_VEL
LIN {X 0,Y 229.204,Z 444.33,A -85,B 0,C 180,E1 -20455.422,E2 -20455.422} C_VEL
LIN {X 0,Y 232.977,Z 435.174,A -85,B 0,C 180,E1 -20458.367,E2 -20458.367} C_VEL
LIN {X 0,Y 236.491,Z 425.85,A -85,B 0,C 180,E1 -20460.84,E2 -20460.84} C_VEL
LIN {X 0,Y 240.872,Z 413.782,A -85,B 0,C 180,E1 -20463.417,E2 -20463.417} C_VEL
LIN {X 0,Y 244.928,Z 401.458,A -85,B 0,C 180,E1 -20465.525,E2 -20465.525} C_VEL
LIN {X 0,Y 248.912,Z 387.857,A -85,B 0,C 180,E1 -20467.377,E2 -20467.377} C_VEL
LIN {X 0,Y 252.233,Z 374.427,A -85,B 0,C 180,E1 -20468.832,E2 -20468.832} C_VEL
LIN {X 0,Y 255.142,Z 359.699,A -85,B 0,C 180,E1 -20470.082,E2 -20470.082} C_VEL
LIN {X 0,Y 257.653,Z 344.14,A -85,B 0,C 180,E1 -20471.022,E2 -20471.022} C_VEL
LIN {X 0,Y 259.359,Z 328.641,A -85,B 0,C 180,E1 -20471.662,E2 -20471.662} C_VEL
LIN {X 0,Y 264.37,Z 238.988,A -85,B 0,C 180,E1 -20473.979,E2 -20473.979} C_VEL
LIN {X 0,Y 257.927,Z 224.644,A -85,B 0,C 180,E1 -20475.939,E2 -20475.939} C_VEL
LIN {X 0,Y 250.666,Z 210.779,A -85,B 0,C 180,E1 -20478.266,E2 -20478.266} C_VEL
LIN {X 0,Y 245.752,Z 202.483,A -85,B 0,C 180,E1 -20479.937,E2 -20479.937} C_VEL
LIN {X 0,Y 239.012,Z 192.785,A -85,B 0,C 180,E1 -20482.367,E2 -20482.367} C_VEL
LIN {X 0,Y 235.43,Z 188.002,A -85,B 0,C 180,E1 -20483.756,E2 -20483.756} C_VEL
LIN {X 0,Y 232.297,Z 183.851,A -85,B 0,C 180,E1 -20485.044,E2 -20485.044} C_VEL
LIN {X 0,Y 229.564,Z 180.274,A -85,B 0,C 180,E1 -20486.231,E2 -20486.231} C_VEL
LIN {X 0,Y 228.63,Z 179.052,A -85,B 0,C 180,E1 -20486.651,E2 -20486.651} C_VEL
LIN {X 0,Y 226.177,Z 176.377,A -85,B 0,C 180,E1 -20487.765,E2 -20487.765} C_VEL
LIN {X 0,Y 224.869,Z 174.137,A -85,B 0,C 180,E1 -20488.432,E2 -20488.432} C_VEL
LIN {X 0,Y 222.466,Z 172.278,A -85,B 0,C 180,E1 -20489.572,E2 -20489.572} C_VEL
LIN {X 0,Y 220.943,Z 169.232,A -85,B 0,C 180,E1 -20490.59,E2 -20490.59} C_VEL
LIN {X 0,Y 220.794,Z 168.634,A -85,B 0,C 180,E1 -20491.22,E2 -20491.22} C_VEL
LIN {X 0,Y 220.857,Z 168.584,A -85,B 0,C 180,E1 -20493.544,E2 -20493.544} C_VEL
LIN {X 0,Y 220.855,Z 168.599,A -85,B 0,C 180,E1 -20497.551,E2 -20497.551} C_VEL
LIN {X 0,Y 220.921,Z 168.59,A -85,B 0,C 180,E1 -20502.625,E2 -20502.625} C_VEL
LIN {X 0,Y 220.989,Z 168.564,A -85,B 0,C 180,E1 -20507.137,E2 -20507.137} C_VEL
LIN {X 0,Y 221.196,Z 168.529,A -85,B 0,C 180,E1 -20510.859,E2 -20510.859} C_VEL
LIN {X 0,Y 221.12,Z 168.566,A -85,B 0,C 180,E1 -20514.528,E2 -20514.528} C_VEL
LIN {X 0,Y 221.474,Z 168.491,A -85,B 0,C 180,E1 -20518.181,E2 -20518.181} C_VEL
LIN {X 0,Y 221.507,Z 168.499,A -85,B 0,C 180,E1 -20521.818,E2 -20521.818} C_VEL
LIN {X 0,Y 221.242,Z 168.544,A -85,B 0,C 180,E1 -20527.3,E2 -20527.3} C_VEL
LIN {X 0,Y 221.089,Z 168.548,A -85,B 0,C 180,E1 -20530.995,E2 -20530.995} C_VEL
LIN {X 0,Y 221.022,Z 168.575,A -85,B 0,C 180,E1 -20532.664,E2 -20532.664} C_VEL
LIN {X 0,Y 220.712,Z 168.627,A -85,B 0,C 180,E1 -20533.682,E2 -20533.682} C_VEL
LIN {X 0,Y 219.339,Z 168.804,A -85,B 0,C 180,E1 -20535.183,E2 -20535.183} C_VEL
LIN {X 0,Y 214.913,Z 169.336,A -85,B 0,C 180,E1 -20538.691,E2 -20538.691} C_VEL
LIN {X 0,Y 213.863,Z 169.448,A -85,B 0,C 180,E1 -20540.268,E2 -20540.268} C_VEL
LIN {X 0,Y 213.79,Z 169.454,A -85,B 0,C 180,E1 -20540.803,E2 -20540.803} C_VEL
LIN {X 0,Y 213.848,Z 169.643,A -85,B 0,C 180,E1 -20545.422,E2 -20545.422} C_VEL
LIN {X 0,Y 214.092,Z 170.682,A -85,B 0,C 180,E1 -20546.109,E2 -20546.109} C_VEL
LIN {X 0,Y 215.612,Z 173.347,A -85,B 0,C 180,E1 -20547.151,E2 -20547.151} C_VEL
LIN {X 0,Y 218.457,Z 175.617,A -85,B 0,C 180,E1 -20548.721,E2 -20548.721} C_VEL
LIN {X 0,Y 220.375,Z 178.74,A -85,B 0,C 180,E1 -20549.818,E2 -20549.818} C_VEL
LIN {X 0,Y 222.798,Z 181.022,A -85,B 0,C 180,E1 -20551.026,E2 -20551.026} C_VEL
LIN {X 0,Y 225.328,Z 184.532,A -85,B 0,C 180,E1 -20552.283,E2 -20552.283} C_VEL
LIN {X 0,Y 226.788,Z 186.127,A -85,B 0,C 180,E1 -20552.952,E2 -20552.952} C_VEL
LIN {X 0,Y 229.718,Z 189.99,A -85,B 0,C 180,E1 -20554.272,E2 -20554.272} C_VEL
LIN {X 0,Y 234.378,Z 196.447,A -85,B 0,C 180,E1 -20556.236,E2 -20556.236} C_VEL
LIN {X 0,Y 240.627,Z 206.626,A -85,B 0,C 180,E1 -20558.694,E2 -20558.694} C_VEL
LIN {X 0,Y 247.269,Z 218.519,A -85,B 0,C 180,E1 -20561.092,E2 -20561.092} C_VEL
LIN {X 0,Y 253.515,Z 231.065,A -85,B 0,C 180,E1 -20563.194,E2 -20563.194} C_VEL
LIN {X 0,Y 259.103,Z 243.823,A -85,B 0,C 180,E1 -20564.984,E2 -20564.984} C_VEL
LIN {X 0,Y 253.996,Z 331.171,A -85,B 0,C 180,E1 -20567.252,E2 -20567.252} C_VEL
LIN {X 0,Y 252.384,Z 346.166,A -85,B 0,C 180,E1 -20567.861,E2 -20567.861} C_VEL
LIN {X 0,Y 250.041,Z 360.247,A -85,B 0,C 180,E1 -20568.66,E2 -20568.66} C_VEL
LIN {X 0,Y 247.232,Z 373.796,A -85,B 0,C 180,E1 -20569.706,E2 -20569.706} C_VEL
LIN {X 0,Y 243.661,Z 388.57,A -85,B 0,C 180,E1 -20571.233,E2 -20571.233} C_VEL
LIN {X 0,Y 239.624,Z 402.312,A -85,B 0,C 180,E1 -20573.04,E2 -20573.04} C_VEL
LIN {X 0,Y 235.249,Z 415.143,A -85,B 0,C 180,E1 -20575.155,E2 -20575.155} C_VEL
LIN {X 0,Y 231.261,Z 425.885,A -85,B 0,C 180,E1 -20577.356,E2 -20577.356} C_VEL
LIN {X 0,Y 226.999,Z 436.71,A -85,B 0,C 180,E1 -20580.099,E2 -20580.099} C_VEL
LIN {X 0,Y 222.873,Z 446.783,A -85,B 0,C 180,E1 -20583.298,E2 -20583.298} C_VEL
LIN {X 0,Y 219.456,Z 454.671,A -85,B 0,C 180,E1 -20586.402,E2 -20586.402} C_VEL
LIN {X 0,Y 216.356,Z 462.038,A -85,B 0,C 180,E1 -20590.058,E2 -20590.058} C_VEL
LIN {X 0,Y 214.172,Z 467.879,A -85,B 0,C 180,E1 -20593.804,E2 -20593.804} C_VEL
LIN {X 0,Y 212.874,Z 471.353,A -85,B 0,C 180,E1 -20596.638,E2 -20596.638} C_VEL
LIN {X 0,Y 211.885,Z 474.862,A -85,B 0,C 180,E1 -20600.454,E2 -20600.454} C_VEL
LIN {X 0,Y 211.405,Z 477.169,A -85,B 0,C 180,E1 -20604.276,E2 -20604.276} C_VEL
LIN {X 0,Y 211.352,Z 478.328,A -85,B 0,C 180,E1 -20608.094,E2 -20608.094} C_VEL
LIN {X 0,Y 211.431,Z 478.48,A -85,B 0,C 180,E1 -20610,E2 -20610} C_VEL
LIN {X 0,Y 211.331,Z 477.85,A -85,B 0,C 180,E1 -20613.91,E2 -20613.91} C_VEL
LIN {X 0,Y 211.596,Z 476.128,A -85,B 0,C 180,E1 -20617.635,E2 -20617.635} C_VEL
LIN {X 0,Y 212.291,Z 473.213,A -85,B 0,C 180,E1 -20621.457,E2 -20621.457} C_VEL
LIN {X 0,Y 213.698,Z 469.064,A -85,B 0,C 180,E1 -20625.254,E2 -20625.254} C_VEL
LIN {X 0,Y 215.847,Z 463.204,A -85,B 0,C 180,E1 -20629.224,E2 -20629.224} C_VEL
LIN {X 0,Y 218.601,Z 456.578,A -85,B 0,C 180,E1 -20632.693,E2 -20632.693} C_VEL
LIN {X 0,Y 222.302,Z 447.881,A -85,B 0,C 180,E1 -20636.27,E2 -20636.27} C_VEL
LIN {X 0,Y 225.4,Z 440.456,A -85,B 0,C 180,E1 -20638.761,E2 -20638.761} C_VEL
LIN {X 0,Y 228.571,Z 432.511,A -85,B 0,C 180,E1 -20640.999,E2 -20640.999} C_VEL
LIN {X 0,Y 232.682,Z 421.989,A -85,B 0,C 180,E1 -20643.451,E2 -20643.451} C_VEL
LIN {X 0,Y 236.771,Z 410.546,A -85,B 0,C 180,E1 -20645.628,E2 -20645.628} C_VEL
LIN {X 0,Y 240.853,Z 398.101,A -85,B 0,C 180,E1 -20647.526,E2 -20647.526} C_VEL
LIN {X 0,Y 244.649,Z 384.46,A -85,B 0,C 180,E1 -20649.197,E2 -20649.197} C_VEL
LIN {X 0,Y 247.892,Z 370.318,A -85,B 0,C 180,E1 -20650.564,E2 -20650.564} C_VEL
LIN {X 0,Y 250.75,Z 355.746,A -85,B 0,C 180,E1 -20651.599,E2 -20651.599} C_VEL
LIN {X 0,Y 252.9,Z 340.762,A -85,B 0,C 180,E1 -20652.369,E2 -20652.369} C_VEL
LIN {X 0,Y 254.298,Z 325.284,A -85,B 0,C 180,E1 -20652.887,E2 -20652.887} C_VEL
LIN {X 0,Y 258.941,Z 244.536,A -85,B 0,C 180,E1 -20654.962,E2 -20654.962} C_VEL
LIN {X 0,Y 258.586,Z 242.805,A -85,B 0,C 180,E1 -20655.107,E2 -20655.107} C_VEL
LIN {X 0,Y 252.342,Z 228.703,A -85,B 0,C 180,E1 -20657.117,E2 -20657.117} C_VEL
LIN {X 0,Y 245.445,Z 215.119,A -85,B 0,C 180,E1 -20659.469,E2 -20659.469} C_VEL
LIN {X 0,Y 237.894,Z 202.134,A -85,B 0,C 180,E1 -20662.26,E2 -20662.26} C_VEL
LIN {X 0,Y 232.819,Z 194.188,A -85,B 0,C 180,E1 -20664.307,E2 -20664.307} C_VEL
LIN {X 0,Y 229.294,Z 189.504,A -85,B 0,C 180,E1 -20665.802,E2 -20665.802} C_VEL
LIN {X 0,Y 226,Z 185.155,A -85,B 0,C 180,E1 -20667.297,E2 -20667.297} C_VEL
LIN {X 0,Y 223.298,Z 181.942,A -85,B 0,C 180,E1 -20668.582,E2 -20668.582} C_VEL
LIN {X 0,Y 222.316,Z 180.444,A -85,B 0,C 180,E1 -20669.089,E2 -20669.089} C_VEL
LIN {X 0,Y 219.698,Z 177.898,A -85,B 0,C 180,E1 -20670.409,E2 -20670.409} C_VEL
LIN {X 0,Y 218.066,Z 175.165,A -85,B 0,C 180,E1 -20671.354,E2 -20671.354} C_VEL
LIN {X 0,Y 215.669,Z 173.426,A -85,B 0,C 180,E1 -20672.66,E2 -20672.66} C_VEL
LIN {X 0,Y 214.198,Z 170.873,A -85,B 0,C 180,E1 -20673.643,E2 -20673.643} C_VEL
LIN {X 0,Y 213.862,Z 169.723,A -85,B 0,C 180,E1 -20674.318,E2 -20674.318} C_VEL
LIN {X 0,Y 213.853,Z 169.462,A -85,B 0,C 180,E1 -20676.953,E2 -20676.953} C_VEL
LIN {X 0,Y 213.945,Z 169.443,A -85,B 0,C 180,E1 -20682.804,E2 -20682.804} C_VEL
LIN {X 0,Y 213.98,Z 169.448,A -85,B 0,C 180,E1 -20686.709,E2 -20686.709} C_VEL
LIN {X 0,Y 214.135,Z 169.406,A -85,B 0,C 180,E1 -20690.555,E2 -20690.555} C_VEL
LIN {X 0,Y 214.086,Z 169.426,A -85,B 0,C 180,E1 -20694.348,E2 -20694.348} C_VEL
LIN {X 0,Y 214.442,Z 169.377,A -85,B 0,C 180,E1 -20698.122,E2 -20698.122} C_VEL
LIN {X 0,Y 214.542,Z 169.376,A -85,B 0,C 180,E1 -20700,E2 -20700} C_VEL
LIN {X 0,Y 214.411,Z 169.37,A -85,B 0,C 180,E1 -20701.879,E2 -20701.879} C_VEL
LIN {X 0,Y 214.183,Z 169.404,A -85,B 0,C 180,E1 -20707.542,E2 -20707.542} C_VEL
LIN {X 0,Y 214.006,Z 169.453,A -85,B 0,C 180,E1 -20711.364,E2 -20711.364} C_VEL
LIN {X 0,Y 213.904,Z 169.439,A -85,B 0,C 180,E1 -20715.239,E2 -20715.239} C_VEL
LIN {X 0,Y 213.796,Z 169.455,A -85,B 0,C 180,E1 -20719.192,E2 -20719.192} C_VEL
LIN {X 0,Y 213.765,Z 169.475,A -85,B 0,C 180,E1 -20723.237,E2 -20723.237} C_VEL
LIN {X 0,Y 213.806,Z 169.721,A -85,B 0,C 180,E1 -20725.885,E2 -20725.885} C_VEL
LIN {X 0,Y 214.139,Z 170.822,A -85,B 0,C 180,E1 -20726.497,E2 -20726.497} C_VEL
LIN {X 0,Y 215.513,Z 173.307,A -85,B 0,C 180,E1 -20727.428,E2 -20727.428} C_VEL
LIN {X 0,Y 218.374,Z 175.547,A -85,B 0,C 180,E1 -20728.996,E2 -20728.996} C_VEL
LIN {X 0,Y 220.283,Z 178.662,A -85,B 0,C 180,E1 -20730.082,E2 -20730.082} C_VEL
LIN {X 0,Y 222.79,Z 181.038,A -85,B 0,C 180,E1 -20731.326,E2 -20731.326} C_VEL
LIN {X 0,Y 225.106,Z 184.398,A -85,B 0,C 180,E1 -20732.481,E2 -20732.481} C_VEL
LIN {X 0,Y 226.748,Z 186.163,A -85,B 0,C 180,E1 -20733.23,E2 -20733.23} C_VEL
LIN {X 0,Y 229.686,Z 189.981,A -85,B 0,C 180,E1 -20734.543,E2 -20734.543} C_VEL
LIN {X 0,Y 234.27,Z 196.334,A -85,B 0,C 180,E1 -20736.468,E2 -20736.468} C_VEL
LIN {X 0,Y 239.545,Z 203.805,A -85,B 0,C 180,E1 -20738.502,E2 -20738.502} C_VEL
LIN {X 0,Y 244.302,Z 211.245,A -85,B 0,C 180,E1 -20740.221,E2 -20740.221} C_VEL
LIN {X 0,Y 250.823,Z 223.326,A -85,B 0,C 180,E1 -20742.462,E2 -20742.462} C_VEL
LIN {X 0,Y 256.984,Z 236.362,A -85,B 0,C 180,E1 -20744.46,E2 -20744.46} C_VEL
LIN {X 0,Y 258.946,Z 240.94,A -85,B 0,C 180,E1 -20745.078,E2 -20745.078} C_VEL
LIN {X 0,Y 257.279,Z 273.463,A -85,B 0,C 180,E1 -20745.958,E2 -20745.958} C_VEL
LIN {X 0,Y 253.887,Z 329.712,A -85,B 0,C 180,E1 -20747.432,E2 -20747.432} C_VEL
LIN {X 0,Y 251.988,Z 345.646,A -85,B 0,C 180,E1 -20748.116,E2 -20748.116} C_VEL
LIN {X 0,Y 249.432,Z 360.779,A -85,B 0,C 180,E1 -20749.073,E2 -20749.073} C_VEL
LIN {X 0,Y 246.279,Z 375.659,A -85,B 0,C 180,E1 -20750.37,E2 -20750.37} C_VEL
LIN {X 0,Y 243.007,Z 388.577,A -85,B 0,C 180,E1 -20751.816,E2 -20751.816} C_VEL
LIN {X 0,Y 238.896,Z 402.054,A -85,B 0,C 180,E1 -20753.697,E2 -20753.697} C_VEL
LIN {X 0,Y 235.078,Z 413.249,A -85,B 0,C 180,E1 -20755.647,E2 -20755.647} C_VEL
LIN {X 0,Y 231.115,Z 423.668,A -85,B 0,C 180,E1 -20757.849,E2 -20757.849} C_VEL
LIN {X 0,Y 227.375,Z 433.334,A -85,B 0,C 180,E1 -20760.36,E2 -20760.36} C_VEL
LIN {X 0,Y 223.357,Z 442.812,A -85,B 0,C 180,E1 -20763.36,E2 -20763.36} C_VEL
LIN {X 0,Y 219.569,Z 451.707,A -85,B 0,C 180,E1 -20766.915,E2 -20766.915} C_VEL
LIN {X 0,Y 216.867,Z 457.927,A -85,B 0,C 180,E1 -20770.019,E2 -20770.019} C_VEL
LIN {X 0,Y 214.575,Z 463.913,A -85,B 0,C 180,E1 -20773.835,E2 -20773.835} C_VEL
LIN {X 0,Y 213.211,Z 467.375,A -85,B 0,C 180,E1 -20776.659,E2 -20776.659} C_VEL
LIN {X 0,Y 212.095,Z 470.878,A -85,B 0,C 180,E1 -20780.463,E2 -20780.463} C_VEL
LIN {X 0,Y 211.514,Z 473.193,A -85,B 0,C 180,E1 -20784.279,E2 -20784.279} C_VEL
LIN {X 0,Y 211.394,Z 474.37,A -85,B 0,C 180,E1 -20788.095,E2 -20788.095} C_VEL
LIN {X 0,Y 211.437,Z 474.527,A -85,B 0,C 180,E1 -20790,E2 -20790} C_VEL
LIN {X 0,Y 211.42,Z 473.852,A -85,B 0,C 180,E1 -20794.241,E2 -20794.241} C_VEL
LIN {X 0,Y 211.721,Z 472.267,A -85,B 0,C 180,E1 -20797.63,E2 -20797.63} C_VEL
LIN {X 0,Y 212.581,Z 469.412,A -85,B 0,C 180,E1 -20801.441,E2 -20801.441} C_VEL
LIN {X 0,Y 214.04,Z 465.325,A -85,B 0,C 180,E1 -20805.229,E2 -20805.229} C_VEL
LIN {X 0,Y 216.185,Z 459.909,A -85,B 0,C 180,E1 -20808.971,E2 -20808.971} C_VEL
LIN {X 0,Y 219.065,Z 453.008,A -85,B 0,C 180,E1 -20812.643,E2 -20812.643} C_VEL
LIN {X 0,Y 222.758,Z 444.395,A -85,B 0,C 180,E1 -20816.213,E2 -20816.213} C_VEL
LIN {X 0,Y 226.685,Z 435.238,A -85,B 0,C 180,E1 -20819.229,E2 -20819.229} C_VEL
LIN {X 0,Y 230.379,Z 425.915,A -85,B 0,C 180,E1 -20821.752,E2 -20821.752} C_VEL
LIN {X 0,Y 234.942,Z 413.846,A -85,B 0,C 180,E1 -20824.376,E2 -20824.376} C_VEL
LIN {X 0,Y 239.176,Z 401.521,A -85,B 0,C 180,E1 -20826.515,E2 -20826.515} C_VEL
LIN {X 0,Y 243.31,Z 387.918,A -85,B 0,C 180,E1 -20828.391,E2 -20828.391} C_VEL
LIN {X 0,Y 246.771,Z 374.269,A -85,B 0,C 180,E1 -20829.891,E2 -20829.891} C_VEL
LIN {X 0,Y 249.763,Z 359.757,A -85,B 0,C 180,E1 -20831.128,E2 -20831.128} C_VEL
LIN {X 0,Y 252.35,Z 344.194,A -85,B 0,C 180,E1 -20832.078,E2 -20832.078} C_VEL
LIN {X 0,Y 254.111,Z 328.688,A -85,B 0,C 180,E1 -20832.724,E2 -20832.724} C_VEL
LIN {X 0,Y 259.225,Z 241.402,A -85,B 0,C 180,E1 -20834.996,E2 -20834.996} C_VEL
LIN {X 0,Y 252.681,Z 226.944,A -85,B 0,C 180,E1 -20837.09,E2 -20837.09} C_VEL
LIN {X 0,Y 245.54,Z 213.277,A -85,B 0,C 180,E1 -20839.517,E2 -20839.517} C_VEL
LIN {X 0,Y 241.396,Z 206.438,A -85,B 0,C 180,E1 -20841.001,E2 -20841.001} C_VEL
LIN {X 0,Y 234.902,Z 197.157,A -85,B 0,C 180,E1 -20843.469,E2 -20843.469} C_VEL
LIN {X 0,Y 231.8,Z 192.925,A -85,B 0,C 180,E1 -20844.74,E2 -20844.74} C_VEL
LIN {X 0,Y 229.265,Z 189.521,A -85,B 0,C 180,E1 -20845.834,E2 -20845.834} C_VEL
LIN {X 0,Y 226.472,Z 185.625,A -85,B 0,C 180,E1 -20847.114,E2 -20847.114} C_VEL
LIN {X 0,Y 223.454,Z 182.182,A -85,B 0,C 180,E1 -20848.54,E2 -20848.54} C_VEL
LIN {X 0,Y 222.381,Z 180.501,A -85,B 0,C 180,E1 -20849.099,E2 -20849.099} C_VEL
LIN {X 0,Y 219.757,Z 177.997,A -85,B 0,C 180,E1 -20850.426,E2 -20850.426} C_VEL
LIN {X 0,Y 218.152,Z 175.214,A -85,B 0,C 180,E1 -20851.366,E2 -20851.366} C_VEL
LIN {X 0,Y 215.579,Z 173.369,A -85,B 0,C 180,E1 -20852.779,E2 -20852.779} C_VEL
LIN {X 0,Y 214.059,Z 170.664,A -85,B 0,C 180,E1 -20853.821,E2 -20853.821} C_VEL
LIN {X 0,Y 213.772,Z 169.582,A -85,B 0,C 180,E1 -20854.567,E2 -20854.567} C_VEL
LIN {X 0,Y 213.776,Z 169.461,A -85,B 0,C 180,E1 -20858.799,E2 -20858.799} C_VEL
LIN {X 0,Y 213.886,Z 169.468,A -85,B 0,C 180,E1 -20862.799,E2 -20862.799} C_VEL
LIN {X 0,Y 213.926,Z 169.439,A -85,B 0,C 180,E1 -20866.705,E2 -20866.705} C_VEL
LIN {X 0,Y 214.136,Z 169.41,A -85,B 0,C 180,E1 -20870.555,E2 -20870.555} C_VEL
LIN {X 0,Y 214.083,Z 169.443,A -85,B 0,C 180,E1 -20874.348,E2 -20874.348} C_VEL
LIN {X 0,Y 214.411,Z 169.37,A -85,B 0,C 180,E1 -20878.121,E2 -20878.121} C_VEL
LIN {X 0,Y 214.539,Z 169.376,A -85,B 0,C 180,E1 -20880,E2 -20880} C_VEL
LIN {X 0,Y 214.44,Z 169.378,A -85,B 0,C 180,E1 -20881.878,E2 -20881.878} C_VEL
LIN {X 0,Y 214.184,Z 169.417,A -85,B 0,C 180,E1 -20887.542,E2 -20887.542} C_VEL
LIN {X 0,Y 214.015,Z 169.433,A -85,B 0,C 180,E1 -20891.363,E2 -20891.363} C_VEL
LIN {X 0,Y 213.935,Z 169.434,A -85,B 0,C 180,E1 -20895.237,E2 -20895.237} C_VEL
LIN {X 0,Y 213.837,Z 169.461,A -85,B 0,C 180,E1 -20899.187,E2 -20899.187} C_VEL
LIN {X 0,Y 213.79,Z 169.454,A -85,B 0,C 180,E1 -20900.803,E2 -20900.803} C_VEL
LIN {X 0,Y 213.8,Z 170.153,A -85,B 0,C 180,E1 -20902.379,E2 -20902.379} C_VEL
LIN {X 0,Y 213.934,Z 172.812,A -85,B 0,C 180,E1 -20904.382,E2 -20904.382} C_VEL
LIN {X 0,Y 214.332,Z 175.728,A -85,B 0,C 180,E1 -20905.791,E2 -20905.791} C_VEL
LIN {X 0,Y 215.569,Z 180.364,A -85,B 0,C 180,E1 -20907.525,E2 -20907.525} C_VEL
LIN {X 0,Y 216.618,Z 182.858,A -85,B 0,C 180,E1 -20908.321,E2 -20908.321} C_VEL
LIN {X 0,Y 219.058,Z 185.993,A -85,B 0,C 180,E1 -20909.685,E2 -20909.685} C_VEL
LIN {X 0,Y 220.546,Z 187.563,A -85,B 0,C 180,E1 -20910.454,E2 -20910.454} C_VEL
LIN {X 0,Y 223.331,Z 191.18,A -85,B 0,C 180,E1 -20911.862,E2 -20911.862} C_VEL
LIN {X 0,Y 228.192,Z 197.714,A -85,B 0,C 180,E1 -20914.133,E2 -20914.133} C_VEL
LIN {X 0,Y 231.719,Z 202.763,A -85,B 0,C 180,E1 -20915.66,E2 -20915.66} C_VEL
LIN {X 0,Y 237.955,Z 213.155,A -85,B 0,C 180,E1 -20918.198,E2 -20918.198} C_VEL
LIN {X 0,Y 244.949,Z 226.232,A -85,B 0,C 180,E1 -20920.806,E2 -20920.806} C_VEL
LIN {X 0,Y 250.917,Z 238.951,A -85,B 0,C 180,E1 -20922.884,E2 -20922.884} C_VEL
LIN {X 0,Y 253.974,Z 246.145,A -85,B 0,C 180,E1 -20923.909,E2 -20923.909} C_VEL
LIN {X 0,Y 248.822,Z 331.123,A -85,B 0,C 180,E1 -20926.141,E2 -20926.141} C_VEL
LIN {X 0,Y 247.161,Z 346.111,A -85,B 0,C 180,E1 -20926.756,E2 -20926.756} C_VEL
LIN {X 0,Y 244.76,Z 360.188,A -85,B 0,C 180,E1 -20927.563,E2 -20927.563} C_VEL
LIN {X 0,Y 241.849,Z 373.735,A -85,B 0,C 180,E1 -20928.616,E2 -20928.616} C_VEL
LIN {X 0,Y 238.244,Z 388.214,A -85,B 0,C 180,E1 -20930.128,E2 -20930.128} C_VEL
LIN {X 0,Y 233.985,Z 402.249,A -85,B 0,C 180,E1 -20931.994,E2 -20931.994} C_VEL
LIN {X 0,Y 229.43,Z 415.079,A -85,B 0,C 180,E1 -20934.137,E2 -20934.137} C_VEL
LIN {X 0,Y 225.282,Z 425.821,A -85,B 0,C 180,E1 -20936.376,E2 -20936.376} C_VEL
LIN {X 0,Y 221.197,Z 435.76,A -85,B 0,C 180,E1 -20938.915,E2 -20938.915} C_VEL
LIN {X 0,Y 217.075,Z 445.484,A -85,B 0,C 180,E1 -20942.001,E2 -20942.001} C_VEL
LIN {X 0,Y 213.377,Z 453.596,A -85,B 0,C 180,E1 -20945.169,E2 -20945.169} C_VEL
LIN {X 0,Y 210.37,Z 460.304,A -85,B 0,C 180,E1 -20948.439,E2 -20948.439} C_VEL
LIN {X 0,Y 207.807,Z 466.498,A -85,B 0,C 180,E1 -20952.279,E2 -20952.279} C_VEL
LIN {X 0,Y 205.921,Z 471.287,A -85,B 0,C 180,E1 -20956.178,E2 -20956.178} C_VEL
LIN {X 0,Y 204.85,Z 474.796,A -85,B 0,C 180,E1 -20960.122,E2 -20960.122} C_VEL
LIN {X 0,Y 204.337,Z 477.103,A -85,B 0,C 180,E1 -20964.077,E2 -20964.077} C_VEL
LIN {X 0,Y 204.26,Z 478.261,A -85,B 0,C 180,E1 -20968.028,E2 -20968.028} C_VEL
LIN {X 0,Y 204.334,Z 478.414,A -85,B 0,C 180,E1 -20970,E2 -20970} C_VEL
LIN {X 0,Y 204.256,Z 477.808,A -85,B 0,C 180,E1 -20973.946,E2 -20973.946} C_VEL
LIN {X 0,Y 204.534,Z 476.061,A -85,B 0,C 180,E1 -20977.9,E2 -20977.9} C_VEL
LIN {X 0,Y 205.299,Z 473.146,A -85,B 0,C 180,E1 -20981.853,E2 -20981.853} C_VEL
LIN {X 0,Y 206.806,Z 468.996,A -85,B 0,C 180,E1 -20985.775,E2 -20985.775} C_VEL
LIN {X 0,Y 208.957,Z 463.5,A -85,B 0,C 180,E1 -20989.654,E2 -20989.654} C_VEL
LIN {X 0,Y 212.013,Z 456.509,A -85,B 0,C 180,E1 -20993.44,E2 -20993.44} C_VEL
LIN {X 0,Y 215.94,Z 447.812,A -85,B 0,C 180,E1 -20997.106,E2 -20997.106} C_VEL
LIN {X 0,Y 219.526,Z 439.252,A -85,B 0,C 180,E1 -21000.037,E2 -21000.037} C_VEL
LIN {X 0,Y 223.855,Z 429.176,A -85,B 0,C 180,E1 -21002.79,E2 -21002.79} C_VEL
LIN {X 0,Y 228.656,Z 416.985,A -85,B 0,C 180,E1 -21005.461,E2 -21005.461} C_VEL
LIN {X 0,Y 233.104,Z 404.549,A -85,B 0,C 180,E1 -21007.628,E2 -21007.628} C_VEL
LIN {X 0,Y 237.254,Z 391.476,A -85,B 0,C 180,E1 -21009.439,E2 -21009.439} C_VEL
LIN {X 0,Y 240.958,Z 377.249,A -85,B 0,C 180,E1 -21011.015,E2 -21011.015} C_VEL
LIN {X 0,Y 243.994,Z 363.466,A -85,B 0,C 180,E1 -21012.182,E2 -21012.182} C_VEL
LIN {X 0,Y 246.734,Z 348.018,A -85,B 0,C 180,E1 -21013.127,E2 -21013.127} C_VEL
LIN {X 0,Y 248.581,Z 332.707,A -85,B 0,C 180,E1 -21013.772,E2 -21013.772} C_VEL
LIN {X 0,Y 253.852,Z 246.468,A -85,B 0,C 180,E1 -21016.04,E2 -21016.04} C_VEL
LIN {X 0,Y 251.813,Z 241.249,A -85,B 0,C 180,E1 -21016.734,E2 -21016.734} C_VEL
LIN {X 0,Y 246.035,Z 228.534,A -85,B 0,C 180,E1 -21018.725,E2 -21018.725} C_VEL
LIN {X 0,Y 240.026,Z 217.023,A -85,B 0,C 180,E1 -21020.913,E2 -21020.913} C_VEL
LIN {X 0,Y 233.002,Z 204.73,A -85,B 0,C 180,E1 -21023.705,E2 -21023.705} C_VEL
LIN {X 0,Y 229.215,Z 199.138,A -85,B 0,C 180,E1 -21025.309,E2 -21025.309} C_VEL
LIN {X 0,Y 226.201,Z 195.083,A -85,B 0,C 180,E1 -21026.653,E2 -21026.653} C_VEL
LIN {X 0,Y 223.475,Z 191.336,A -85,B 0,C 180,E1 -21027.948,E2 -21027.948} C_VEL
LIN {X 0,Y 220.543,Z 187.64,A -85,B 0,C 180,E1 -21029.412,E2 -21029.412} C_VEL
LIN {X 0,Y 219.653,Z 186.531,A -85,B 0,C 180,E1 -21029.876,E2 -21029.876} C_VEL
LIN {X 0,Y 217.053,Z 183.588,A -85,B 0,C 180,E1 -21031.274,E2 -21031.274} C_VEL
LIN {X 0,Y 215.897,Z 181.691,A -85,B 0,C 180,E1 -21031.967,E2 -21031.967} C_VEL
LIN {X 0,Y 213.294,Z 179.43,A -85,B 0,C 180,E1 -21033.471,E2 -21033.471} C_VEL
LIN {X 0,Y 211.541,Z 176.302,A -85,B 0,C 180,E1 -21034.676,E2 -21034.676} C_VEL
LIN {X 0,Y 208.775,Z 174.462,A -85,B 0,C 180,E1 -21036.478,E2 -21036.478} C_VEL
LIN {X 0,Y 207.087,Z 171.748,A -85,B 0,C 180,E1 -21037.845,E2 -21037.845} C_VEL
LIN {X 0,Y 206.806,Z 170.633,A -85,B 0,C 180,E1 -21038.573,E2 -21038.573} C_VEL
LIN {X 0,Y 206.875,Z 170.333,A -85,B 0,C 180,E1 -21042.197,E2 -21042.197} C_VEL
LIN {X 0,Y 206.914,Z 170.32,A -85,B 0,C 180,E1 -21046.246,E2 -21046.246} C_VEL
LIN {X 0,Y 207.079,Z 170.284,A -85,B 0,C 180,E1 -21050.23,E2 -21050.23} C_VEL
LIN {X 0,Y 207.048,Z 170.304,A -85,B 0,C 180,E1 -21054.156,E2 -21054.156} C_VEL
LIN {X 0,Y 207.378,Z 170.255,A -85,B 0,C 180,E1 -21058.058,E2 -21058.058} C_VEL
LIN {X 0,Y 207.506,Z 170.251,A -85,B 0,C 180,E1 -21060,E2 -21060} C_VEL
LIN {X 0,Y 207.052,Z 170.293,A -85,B 0,C 180,E1 -21063.893,E2 -21063.893} C_VEL
LIN {X 0,Y 207.128,Z 170.28,A -85,B 0,C 180,E1 -21067.801,E2 -21067.801} C_VEL
LIN {X 0,Y 206.928,Z 170.334,A -85,B 0,C 180,E1 -21071.758,E2 -21071.758} C_VEL
LIN {X 0,Y 206.829,Z 170.324,A -85,B 0,C 180,E1 -21075.774,E2 -21075.774} C_VEL
LIN {X 0,Y 206.715,Z 170.333,A -85,B 0,C 180,E1 -21079.876,E2 -21079.876} C_VEL
LIN {X 0,Y 206.788,Z 170.728,A -85,B 0,C 180,E1 -21081.691,E2 -21081.691} C_VEL
LIN {X 0,Y 207.138,Z 172.003,A -85,B 0,C 180,E1 -21082.399,E2 -21082.399} C_VEL
LIN {X 0,Y 208.773,Z 174.559,A -85,B 0,C 180,E1 -21083.706,E2 -21083.706} C_VEL
LIN {X 0,Y 211.642,Z 176.524,A -85,B 0,C 180,E1 -21085.575,E2 -21085.575} C_VEL
LIN {X 0,Y 213.277,Z 179.48,A -85,B 0,C 180,E1 -21086.7,E2 -21086.7} C_VEL
LIN {X 0,Y 216.215,Z 182.193,A -85,B 0,C 180,E1 -21088.401,E2 -21088.401} C_VEL
LIN {X 0,Y 218.433,Z 185.437,A -85,B 0,C 180,E1 -21089.675,E2 -21089.675} C_VEL
LIN {X 0,Y 220.284,Z 187.221,A -85,B 0,C 180,E1 -21090.625,E2 -21090.625} C_VEL
LIN {X 0,Y 223.082,Z 191.025,A -85,B 0,C 180,E1 -21092.049,E2 -21092.049} C_VEL
LIN {X 0,Y 224.738,Z 193.202,A -85,B 0,C 180,E1 -21092.846,E2 -21092.846} C_VEL
LIN {X 0,Y 228.102,Z 197.653,A -85,B 0,C 180,E1 -21094.381,E2 -21094.381} C_VEL
LIN {X 0,Y 233.525,Z 205.212,A -85,B 0,C 180,E1 -21096.67,E2 -21096.67} C_VEL
LIN {X 0,Y 240.074,Z 215.169,A -85,B 0,C 180,E1 -21099.192,E2 -21099.192} C_VEL
LIN {X 0,Y 246.604,Z 227.59,A -85,B 0,C 180,E1 -21101.561,E2 -21101.561} C_VEL
LIN {X 0,Y 252.107,Z 239.3,A -85,B 0,C 180,E1 -21103.435,E2 -21103.435} C_VEL
LIN {X 0,Y 253.922,Z 243.462,A -85,B 0,C 180,E1 -21104.033,E2 -21104.033} C_VEL
LIN {X 0,Y 248.722,Z 329.794,A -85,B 0,C 180,E1 -21106.329,E2 -21106.329} C_VEL
LIN {X 0,Y 246.767,Z 345.722,A -85,B 0,C 180,E1 -21107.02,E2 -21107.02} C_VEL
LIN {X 0,Y 244.122,Z 360.852,A -85,B 0,C 180,E1 -21107.984,E2 -21107.984} C_VEL
LIN {X 0,Y 240.898,Z 375.574,A -85,B 0,C 180,E1 -21109.277,E2 -21109.277} C_VEL
LIN {X 0,Y 237.473,Z 388.648,A -85,B 0,C 180,E1 -21110.758,E2 -21110.758} C_VEL
LIN {X 0,Y 233.207,Z 402.125,A -85,B 0,C 180,E1 -21112.664,E2 -21112.664} C_VEL
LIN {X 0,Y 229.223,Z 413.319,A -85,B 0,C 180,E1 -21114.64,E2 -21114.64} C_VEL
LIN {X 0,Y 225.11,Z 423.738,A -85,B 0,C 180,E1 -21116.883,E2 -21116.883} C_VEL
LIN {X 0,Y 221.17,Z 433.403,A -85,B 0,C 180,E1 -21119.441,E2 -21119.441} C_VEL
LIN {X 0,Y 217.569,Z 441.654,A -85,B 0,C 180,E1 -21122.071,E2 -21122.071} C_VEL
LIN {X 0,Y 213.938,Z 449.766,A -85,B 0,C 180,E1 -21125.238,E2 -21125.238} C_VEL
LIN {X 0,Y 210.875,Z 456.461,A -85,B 0,C 180,E1 -21128.494,E2 -21128.494} C_VEL
LIN {X 0,Y 208.267,Z 462.658,A -85,B 0,C 180,E1 -21132.32,E2 -21132.32} C_VEL
LIN {X 0,Y 206.258,Z 467.443,A -85,B 0,C 180,E1 -21136.201,E2 -21136.201} C_VEL
LIN {X 0,Y 205.08,Z 470.945,A -85,B 0,C 180,E1 -21140.134,E2 -21140.134} C_VEL
LIN {X 0,Y 204.444,Z 473.259,A -85,B 0,C 180,E1 -21144.081,E2 -21144.081} C_VEL
LIN {X 0,Y 204.302,Z 474.437,A -85,B 0,C 180,E1 -21148.029,E2 -21148.029} C_VEL
LIN {X 0,Y 204.342,Z 474.594,A -85,B 0,C 180,E1 -21150,E2 -21150} C_VEL
LIN {X 0,Y 204.322,Z 474.001,A -85,B 0,C 180,E1 -21154.045,E2 -21154.045} C_VEL
LIN {X 0,Y 204.666,Z 472.333,A -85,B 0,C 180,E1 -21157.895,E2 -21157.895} C_VEL
LIN {X 0,Y 205.574,Z 469.478,A -85,B 0,C 180,E1 -21161.837,E2 -21161.837} C_VEL
LIN {X 0,Y 207.173,Z 465.391,A -85,B 0,C 180,E1 -21165.747,E2 -21165.747} C_VEL
LIN {X 0,Y 209.446,Z 459.974,A -85,B 0,C 180,E1 -21169.606,E2 -21169.606} C_VEL
LIN {X 0,Y 212.496,Z 453.073,A -85,B 0,C 180,E1 -21173.384,E2 -21173.384} C_VEL
LIN {X 0,Y 216.367,Z 444.46,A -85,B 0,C 180,E1 -21177.049,E2 -21177.049} C_VEL
LIN {X 0,Y 219.916,Z 436.716,A -85,B 0,C 180,E1 -21179.693,E2 -21179.693} C_VEL
LIN {X 0,Y 223.66,Z 427.603,A -85,B 0,C 180,E1 -21182.289,E2 -21182.289} C_VEL
LIN {X 0,Y 227.974,Z 416.851,A -85,B 0,C 180,E1 -21184.773,E2 -21184.773} C_VEL
LIN {X 0,Y 232.294,Z 405.114,A -85,B 0,C 180,E1 -21186.964,E2 -21186.964} C_VEL
LIN {X 0,Y 236.423,Z 392.367,A -85,B 0,C 180,E1 -21188.887,E2 -21188.887} C_VEL
LIN {X 0,Y 240.412,Z 378.153,A -85,B 0,C 180,E1 -21190.574,E2 -21190.574} C_VEL
LIN {X 0,Y 243.503,Z 364.355,A -85,B 0,C 180,E1 -21191.87,E2 -21191.87} C_VEL
LIN {X 0,Y 246.256,Z 349.679,A -85,B 0,C 180,E1 -21192.882,E2 -21192.882} C_VEL
LIN {X 0,Y 248.346,Z 334.595,A -85,B 0,C 180,E1 -21193.614,E2 -21193.614} C_VEL
LIN {X 0,Y 249.735,Z 317.512,A -85,B 0,C 180,E1 -21194.148,E2 -21194.148} C_VEL
LIN {X 0,Y 254.121,Z 243.715,A -85,B 0,C 180,E1 -21196.067,E2 -21196.067} C_VEL
LIN {X 0,Y 247.666,Z 229.564,A -85,B 0,C 180,E1 -21198.243,E2 -21198.243} C_VEL
LIN {X 0,Y 241.039,Z 216.854,A -85,B 0,C 180,E1 -21200.624,E2 -21200.624} C_VEL
LIN {X 0,Y 236.392,Z 209.397,A -85,B 0,C 180,E1 -21202.381,E2 -21202.381} C_VEL
LIN {X 0,Y 230.03,Z 200.141,A -85,B 0,C 180,E1 -21204.983,E2 -21204.983} C_VEL
LIN {X 0,Y 226.028,Z 194.869,A -85,B 0,C 180,E1 -21206.759,E2 -21206.759} C_VEL
LIN {X 0,Y 223.27,Z 191.109,A -85,B 0,C 180,E1 -21208.08,E2 -21208.08} C_VEL
LIN {X 0,Y 220.512,Z 187.565,A -85,B 0,C 180,E1 -21209.474,E2 -21209.474} C_VEL
LIN {X 0,Y 219.404,Z 186.353,A -85,B 0,C 180,E1 -21210.047,E2 -21210.047} C_VEL
LIN {X 0,Y 216.769,Z 183.176,A -85,B 0,C 180,E1 -21211.497,E2 -21211.497} C_VEL
LIN {X 0,Y 215.794,Z 181.649,A -85,B 0,C 180,E1 -21212.084,E2 -21212.084} C_VEL
LIN {X 0,Y 213.292,Z 179.452,A -85,B 0,C 180,E1 -21213.546,E2 -21213.546} C_VEL
LIN {X 0,Y 211.303,Z 176.193,A -85,B 0,C 180,E1 -21214.908,E2 -21214.908} C_VEL
LIN {X 0,Y 208.67,Z 174.429,A -85,B 0,C 180,E1 -21216.652,E2 -21216.652} C_VEL
LIN {X 0,Y 207.104,Z 171.913,A -85,B 0,C 180,E1 -21217.933,E2 -21217.933} C_VEL
LIN {X 0,Y 206.79,Z 170.642,A -85,B 0,C 180,E1 -21218.701,E2 -21218.701} C_VEL
LIN {X 0,Y 206.823,Z 170.337,A -85,B 0,C 180,E1 -21222.192,E2 -21222.192} C_VEL
LIN {X 0,Y 206.866,Z 170.314,A -85,B 0,C 180,E1 -21226.242,E2 -21226.242} C_VEL
LIN {X 0,Y 207.08,Z 170.291,A -85,B 0,C 180,E1 -21230.23,E2 -21230.23} C_VEL
LIN {X 0,Y 207.045,Z 170.316,A -85,B 0,C 180,E1 -21234.155,E2 -21234.155} C_VEL
LIN {X 0,Y 207.35,Z 170.249,A -85,B 0,C 180,E1 -21238.057,E2 -21238.057} C_VEL
LIN {X 0,Y 207.504,Z 170.251,A -85,B 0,C 180,E1 -21240,E2 -21240} C_VEL
LIN {X 0,Y 207.376,Z 170.255,A -85,B 0,C 180,E1 -21241.942,E2 -21241.942} C_VEL
LIN {X 0,Y 207.128,Z 170.291,A -85,B 0,C 180,E1 -21247.8,E2 -21247.8} C_VEL
LIN {X 0,Y 206.944,Z 170.319,A -85,B 0,C 180,E1 -21251.757,E2 -21251.757} C_VEL
LIN {X 0,Y 206.868,Z 170.314,A -85,B 0,C 180,E1 -21255.77,E2 -21255.77} C_VEL
LIN {X 0,Y 206.764,Z 170.337,A -85,B 0,C 180,E1 -21259.871,E2 -21259.871} C_VEL
LIN {X 0,Y 206.808,Z 170.596,A -85,B 0,C 180,E1 -21261.166,E2 -21261.166} C_VEL
LIN {X 0,Y 207.065,Z 171.676,A -85,B 0,C 180,E1 -21261.922,E2 -21261.922} C_VEL
LIN {X 0,Y 208.333,Z 173.973,A -85,B 0,C 180,E1 -21263.006,E2 -21263.006} C_VEL
LIN {X 0,Y 210.713,Z 175.939,A -85,B 0,C 180,E1 -21264.64,E2 -21264.64} C_VEL
LIN {X 0,Y 211.667,Z 176.54,A -85,B 0,C 180,E1 -21265.242,E2 -21265.242} C_VEL
LIN {X 0,Y 213.588,Z 179.77,A -85,B 0,C 180,E1 -21266.551,E2 -21266.551} C_VEL
LIN {X 0,Y 216.28,Z 182.214,A -85,B 0,C 180,E1 -21268.11,E2 -21268.11} C_VEL
LIN {X 0,Y 216.618,Z 182.858,A -85,B 0,C 180,E1 -21268.321,E2 -21268.321} C_VEL
LIN {X 0,Y 217.99,Z 186.686,A -85,B 0,C 180,E1 -21269.236,E2 -21269.236} C_VEL
LIN {X 0,Y 220.621,Z 196.248,A -85,B 0,C 180,E1 -21271.028,E2 -21271.028} C_VEL
LIN {X 0,Y 221.924,Z 198.818,A -85,B 0,C 180,E1 -21271.737,E2 -21271.737} C_VEL
LIN {X 0,Y 226.498,Z 205.148,A -85,B 0,C 180,E1 -21273.912,E2 -21273.912} C_VEL
LIN {X 0,Y 229.925,Z 210.38,A -85,B 0,C 180,E1 -21275.437,E2 -21275.437} C_VEL
LIN {X 0,Y 236.084,Z 221.292,A -85,B 0,C 180,E1 -21278.013,E2 -21278.013} C_VEL
LIN {X 0,Y 242.46,Z 233.827,A -85,B 0,C 180,E1 -21280.462,E2 -21280.462} C_VEL
LIN {X 0,Y 248.082,Z 246.443,A -85,B 0,C 180,E1 -21282.491,E2 -21282.491} C_VEL
LIN {X 0,Y 248.988,Z 248.635,A -85,B 0,C 180,E1 -21282.809,E2 -21282.809} C_VEL
LIN {X 0,Y 243.765,Z 331.075,A -85,B 0,C 180,E1 -21284.987,E2 -21284.987} C_VEL
LIN {X 0,Y 242.044,Z 346.056,A -85,B 0,C 180,E1 -21285.606,E2 -21285.606} C_VEL
LIN {X 0,Y 239.58,Z 360.13,A -85,B 0,C 180,E1 -21286.42,E2 -21286.42} C_VEL
LIN {X 0,Y 236.568,Z 373.675,A -85,B 0,C 180,E1 -21287.479,E2 -21287.479} C_VEL
LIN {X 0,Y 232.919,Z 387.834,A -85,B 0,C 180,E1 -21288.967,E2 -21288.967} C_VEL
LIN {X 0,Y 228.857,Z 400.895,A -85,B 0,C 180,E1 -21290.7,E2 -21290.7} C_VEL
LIN {X 0,Y 224.11,Z 413.946,A -85,B 0,C 180,E1 -21292.866,E2 -21292.866} C_VEL
LIN {X 0,Y 219.37,Z 425.757,A -85,B 0,C 180,E1 -21295.343,E2 -21295.343} C_VEL
LIN {X 0,Y 215.095,Z 435.695,A -85,B 0,C 180,E1 -21297.93,E2 -21297.93} C_VEL
LIN {X 0,Y 210.774,Z 445.419,A -85,B 0,C 180,E1 -21301.087,E2 -21301.087} C_VEL
LIN {X 0,Y 206.903,Z 453.53,A -85,B 0,C 180,E1 -21304.336,E2 -21304.336} C_VEL
LIN {X 0,Y 203.718,Z 460.239,A -85,B 0,C 180,E1 -21307.698,E2 -21307.698} C_VEL
LIN {X 0,Y 201,Z 466.432,A -85,B 0,C 180,E1 -21311.658,E2 -21311.658} C_VEL
LIN {X 0,Y 198.989,Z 471.221,A -85,B 0,C 180,E1 -21315.686,E2 -21315.686} C_VEL
LIN {X 0,Y 197.833,Z 474.73,A -85,B 0,C 180,E1 -21319.768,E2 -21319.768} C_VEL
LIN {X 0,Y 197.268,Z 477.037,A -85,B 0,C 180,E1 -21323.864,E2 -21323.864} C_VEL
LIN {X 0,Y 197.171,Z 478.195,A -85,B 0,C 180,E1 -21327.957,E2 -21327.957} C_VEL
LIN {X 0,Y 197.24,Z 478.348,A -85,B 0,C 180,E1 -21330,E2 -21330} C_VEL
LIN {X 0,Y 197.171,Z 477.742,A -85,B 0,C 180,E1 -21334.088,E2 -21334.088} C_VEL
LIN {X 0,Y 197.472,Z 475.993,A -85,B 0,C 180,E1 -21338.184,E2 -21338.184} C_VEL
LIN {X 0,Y 198.304,Z 473.078,A -85,B 0,C 180,E1 -21342.277,E2 -21342.277} C_VEL
LIN {X 0,Y 199.933,Z 468.929,A -85,B 0,C 180,E1 -21346.333,E2 -21346.333} C_VEL
LIN {X 0,Y 202.213,Z 463.432,A -85,B 0,C 180,E1 -21350.338,E2 -21350.338} C_VEL
LIN {X 0,Y 205.446,Z 456.441,A -85,B 0,C 180,E1 -21354.236,E2 -21354.236} C_VEL
LIN {X 0,Y 209.001,Z 448.964,A -85,B 0,C 180,E1 -21357.54,E2 -21357.54} C_VEL
LIN {X 0,Y 212.515,Z 441.245,A -85,B 0,C 180,E1 -21360.31,E2 -21360.31} C_VEL
LIN {X 0,Y 215.722,Z 434.002,A -85,B 0,C 180,E1 -21362.517,E2 -21362.517} C_VEL
LIN {X 0,Y 220.15,Z 423.768,A -85,B 0,C 180,E1 -21365.073,E2 -21365.073} C_VEL
LIN {X 0,Y 224.929,Z 411.561,A -85,B 0,C 180,E1 -21367.538,E2 -21367.538} C_VEL
LIN {X 0,Y 229.733,Z 397.96,A -85,B 0,C 180,E1 -21369.688,E2 -21369.688} C_VEL
LIN {X 0,Y 233.789,Z 384.316,A -85,B 0,C 180,E1 -21371.403,E2 -21371.403} C_VEL
LIN {X 0,Y 237.29,Z 370.171,A -85,B 0,C 180,E1 -21372.793,E2 -21372.793} C_VEL
LIN {X 0,Y 240.335,Z 355.596,A -85,B 0,C 180,E1 -21373.843,E2 -21373.843} C_VEL
LIN {X 0,Y 242.614,Z 340.606,A -85,B 0,C 180,E1 -21374.625,E2 -21374.625} C_VEL
LIN {X 0,Y 244.079,Z 325.111,A -85,B 0,C 180,E1 -21375.158,E2 -21375.158} C_VEL
LIN {X 0,Y 248.79,Z 248.413,A -85,B 0,C 180,E1 -21377.178,E2 -21377.178} C_VEL
LIN {X 0,Y 243.086,Z 235.279,A -85,B 0,C 180,E1 -21379.222,E2 -21379.222} C_VEL
LIN {X 0,Y 236.731,Z 222.577,A -85,B 0,C 180,E1 -21381.636,E2 -21381.636} C_VEL
LIN {X 0,Y 229.645,Z 209.959,A -85,B 0,C 180,E1 -21384.581,E2 -21384.581} C_VEL
LIN {X 0,Y 226.192,Z 204.728,A -85,B 0,C 180,E1 -21386.116,E2 -21386.116} C_VEL
LIN {X 0,Y 223.243,Z 200.679,A -85,B 0,C 180,E1 -21387.492,E2 -21387.492} C_VEL
LIN {X 0,Y 220.568,Z 197.058,A -85,B 0,C 180,E1 -21388.817,E2 -21388.817} C_VEL
LIN {X 0,Y 217.248,Z 192.719,A -85,B 0,C 180,E1 -21390.574,E2 -21390.574} C_VEL
LIN {X 0,Y 214.575,Z 189.49,A -85,B 0,C 180,E1 -21392.086,E2 -21392.086} C_VEL
LIN {X 0,Y 213.565,Z 188.029,A -85,B 0,C 180,E1 -21392.704,E2 -21392.704} C_VEL
LIN {X 0,Y 210.921,Z 185.323,A -85,B 0,C 180,E1 -21394.331,E2 -21394.331} C_VEL
LIN {X 0,Y 209.332,Z 182.791,A -85,B 0,C 180,E1 -21395.451,E2 -21395.451} C_VEL
LIN {X 0,Y 206.646,Z 180.58,A -85,B 0,C 180,E1 -21397.323,E2 -21397.323} C_VEL
LIN {X 0,Y 204.521,Z 177.147,A -85,B 0,C 180,E1 -21399.114,E2 -21399.114} C_VEL
LIN {X 0,Y 201.659,Z 175.185,A -85,B 0,C 180,E1 -21401.563,E2 -21401.563} C_VEL
LIN {X 0,Y 200.081,Z 172.453,A -85,B 0,C 180,E1 -21403.352,E2 -21403.352} C_VEL
LIN {X 0,Y 199.872,Z 171.419,A -85,B 0,C 180,E1 -21404.448,E2 -21404.448} C_VEL
LIN {X 0,Y 200.024,Z 171.163,A -85,B 0,C 180,E1 -21409.882,E2 -21409.882} C_VEL
LIN {X 0,Y 200.01,Z 171.183,A -85,B 0,C 180,E1 -21413.949,E2 -21413.949} C_VEL
LIN {X 0,Y 200.317,Z 171.132,A -85,B 0,C 180,E1 -21417.99,E2 -21417.99} C_VEL
LIN {X 0,Y 200.471,Z 171.126,A -85,B 0,C 180,E1 -21420,E2 -21420} C_VEL
LIN {X 0,Y 199.998,Z 171.173,A -85,B 0,C 180,E1 -21424.03,E2 -21424.03} C_VEL
LIN {X 0,Y 200.076,Z 171.157,A -85,B 0,C 180,E1 -21428.077,E2 -21428.077} C_VEL
LIN {X 0,Y 199.874,Z 171.203,A -85,B 0,C 180,E1 -21432.18,E2 -21432.18} C_VEL
LIN {X 0,Y 199.837,Z 171.485,A -85,B 0,C 180,E1 -21435.882,E2 -21435.882} C_VEL
LIN {X 0,Y 200.116,Z 172.698,A -85,B 0,C 180,E1 -21436.908,E2 -21436.908} C_VEL
LIN {X 0,Y 201.832,Z 175.47,A -85,B 0,C 180,E1 -21438.79,E2 -21438.79} C_VEL
LIN {X 0,Y 204.824,Z 177.487,A -85,B 0,C 180,E1 -21441.315,E2 -21441.315} C_VEL
LIN {X 0,Y 206.65,Z 180.714,A -85,B 0,C 180,E1 -21442.868,E2 -21442.868} C_VEL
LIN {X 0,Y 209.1,Z 182.698,A -85,B 0,C 180,E1 -21444.578,E2 -21444.578} C_VEL
LIN {X 0,Y 209.751,Z 183.44,A -85,B 0,C 180,E1 -21445.025,E2 -21445.025} C_VEL
LIN {X 0,Y 211.903,Z 186.611,A -85,B 0,C 180,E1 -21446.487,E2 -21446.487} C_VEL
LIN {X 0,Y 213.957,Z 188.531,A -85,B 0,C 180,E1 -21447.71,E2 -21447.71} C_VEL
LIN {X 0,Y 216.596,Z 192.144,A -85,B 0,C 180,E1 -21449.258,E2 -21449.258} C_VEL
LIN {X 0,Y 218.051,Z 193.74,A -85,B 0,C 180,E1 -21450.039,E2 -21450.039} C_VEL
LIN {X 0,Y 222.129,Z 199.241,A -85,B 0,C 180,E1 -21452.147,E2 -21452.147} C_VEL
LIN {X 0,Y 225.776,Z 204.229,A -85,B 0,C 180,E1 -21453.876,E2 -21453.876} C_VEL
LIN {X 0,Y 230.385,Z 210.732,A -85,B 0,C 180,E1 -21455.893,E2 -21455.893} C_VEL
LIN {X 0,Y 236.703,Z 220.673,A -85,B 0,C 180,E1 -21458.441,E2 -21458.441} C_VEL
LIN {X 0,Y 242.789,Z 232.48,A -85,B 0,C 180,E1 -21460.749,E2 -21460.749} C_VEL
LIN {X 0,Y 247.856,Z 243.502,A -85,B 0,C 180,E1 -21462.56,E2 -21462.56} C_VEL
LIN {X 0,Y 248.904,Z 245.924,A -85,B 0,C 180,E1 -21462.924,E2 -21462.924} C_VEL
LIN {X 0,Y 243.65,Z 329.876,A -85,B 0,C 180,E1 -21465.179,E2 -21465.179} C_VEL
LIN {X 0,Y 241.741,Z 345.023,A -85,B 0,C 180,E1 -21465.827,E2 -21465.827} C_VEL
LIN {X 0,Y 238.893,Z 360.926,A -85,B 0,C 180,E1 -21466.844,E2 -21466.844} C_VEL
LIN {X 0,Y 235.891,Z 374.381,A -85,B 0,C 180,E1 -21468.021,E2 -21468.021} C_VEL
LIN {X 0,Y 231.991,Z 388.817,A -85,B 0,C 180,E1 -21469.663,E2 -21469.663} C_VEL
LIN {X 0,Y 227.599,Z 402.195,A -85,B 0,C 180,E1 -21471.579,E2 -21471.579} C_VEL
LIN {X 0,Y 223.057,Z 414.429,A -85,B 0,C 180,E1 -21473.788,E2 -21473.788} C_VEL
LIN {X 0,Y 218.432,Z 425.579,A -85,B 0,C 180,E1 -21476.288,E2 -21476.288} C_VEL
LIN {X 0,Y 214.423,Z 434.954,A -85,B 0,C 180,E1 -21478.92,E2 -21478.92} C_VEL
LIN {X 0,Y 210.096,Z 444.177,A -85,B 0,C 180,E1 -21482.075,E2 -21482.075} C_VEL
LIN {X 0,Y 206.487,Z 451.844,A -85,B 0,C 180,E1 -21485.358,E2 -21485.358} C_VEL
LIN {X 0,Y 203.14,Z 458.792,A -85,B 0,C 180,E1 -21489.086,E2 -21489.086} C_VEL
LIN {X 0,Y 200.88,Z 464.049,A -85,B 0,C 180,E1 -21492.7,E2 -21492.7} C_VEL
LIN {X 0,Y 199.327,Z 467.51,A -85,B 0,C 180,E1 -21495.711,E2 -21495.711} C_VEL
LIN {X 0,Y 198.049,Z 471.013,A -85,B 0,C 180,E1 -21499.78,E2 -21499.78} C_VEL
LIN {X 0,Y 197.371,Z 473.326,A -85,B 0,C 180,E1 -21503.868,E2 -21503.868} C_VEL
LIN {X 0,Y 197.213,Z 474.503,A -85,B 0,C 180,E1 -21507.958,E2 -21507.958} C_VEL
LIN {X 0,Y 197.248,Z 474.66,A -85,B 0,C 180,E1 -21510,E2 -21510} C_VEL
LIN {X 0,Y 197.246,Z 474.091,A -85,B 0,C 180,E1 -21514.087,E2 -21514.087} C_VEL
LIN {X 0,Y 197.632,Z 472.399,A -85,B 0,C 180,E1 -21518.178,E2 -21518.178} C_VEL
LIN {X 0,Y 198.584,Z 469.544,A -85,B 0,C 180,E1 -21522.26,E2 -21522.26} C_VEL
LIN {X 0,Y 200.293,Z 465.457,A -85,B 0,C 180,E1 -21526.303,E2 -21526.303} C_VEL
LIN {X 0,Y 202.71,Z 460.04,A -85,B 0,C 180,E1 -21530.286,E2 -21530.286} C_VEL
LIN {X 0,Y 205.941,Z 453.138,A -85,B 0,C 180,E1 -21534.175,E2 -21534.175} C_VEL
LIN {X 0,Y 210.03,Z 444.525,A -85,B 0,C 180,E1 -21537.935,E2 -21537.935} C_VEL
LIN {X 0,Y 213.71,Z 436.781,A -85,B 0,C 180,E1 -21540.646,E2 -21540.646} C_VEL
LIN {X 0,Y 217.659,Z 427.667,A -85,B 0,C 180,E1 -21543.293,E2 -21543.293} C_VEL
LIN {X 0,Y 222.157,Z 416.914,A -85,B 0,C 180,E1 -21545.821,E2 -21545.821} C_VEL
LIN {X 0,Y 226.619,Z 405.177,A -85,B 0,C 180,E1 -21548.052,E2 -21548.052} C_VEL
LIN {X 0,Y 230.907,Z 392.517,A -85,B 0,C 180,E1 -21549.982,E2 -21549.982} C_VEL
LIN {X 0,Y 234.882,Z 378.877,A -85,B 0,C 180,E1 -21551.631,E2 -21551.631} C_VEL
LIN {X 0,Y 238.261,Z 364.414,A -85,B 0,C 180,E1 -21553.01,E2 -21553.01} C_VEL
LIN {X 0,Y 241.242,Z 348.973,A -85,B 0,C 180,E1 -21554.07,E2 -21554.07} C_VEL
LIN {X 0,Y 243.39,Z 333.507,A -85,B 0,C 180,E1 -21554.809,E2 -21554.809} C_VEL
LIN {X 0,Y 244.934,Z 313.978,A -85,B 0,C 180,E1 -21555.394,E2 -21555.394} C_VEL
LIN {X 0,Y 249.046,Z 246.13,A -85,B 0,C 180,E1 -21557.194,E2 -21557.194} C_VEL
LIN {X 0,Y 243.317,Z 233.362,A -85,B 0,C 180,E1 -21559.237,E2 -21559.237} C_VEL
LIN {X 0,Y 236.899,Z 220.903,A -85,B 0,C 180,E1 -21561.668,E2 -21561.668} C_VEL
LIN {X 0,Y 231.616,Z 212.569,A -85,B 0,C 180,E1 -21563.781,E2 -21563.781} C_VEL
LIN {X 0,Y 226.267,Z 204.833,A -85,B 0,C 180,E1 -21566.106,E2 -21566.106} C_VEL
LIN {X 0,Y 223.318,Z 200.794,A -85,B 0,C 180,E1 -21567.488,E2 -21567.488} C_VEL
LIN {X 0,Y 220.632,Z 197.125,A -85,B 0,C 180,E1 -21568.827,E2 -21568.827} C_VEL
LIN {X 0,Y 217.319,Z 192.818,A -85,B 0,C 180,E1 -21570.588,E2 -21570.588} C_VEL
LIN {X 0,Y 214.465,Z 189.348,A -85,B 0,C 180,E1 -21572.215,E2 -21572.215} C_VEL
LIN {X 0,Y 213.498,Z 187.974,A -85,B 0,C 180,E1 -21572.812,E2 -21572.812} C_VEL
LIN {X 0,Y 210.939,Z 185.392,A -85,B 0,C 180,E1 -21574.4,E2 -21574.4} C_VEL
LIN {X 0,Y 209.455,Z 182.869,A -85,B 0,C 180,E1 -21575.466,E2 -21575.466} C_VEL
LIN {X 0,Y 206.815,Z 180.855,A -85,B 0,C 180,E1 -21577.301,E2 -21577.301} C_VEL
LIN {X 0,Y 204.992,Z 177.901,A -85,B 0,C 180,E1 -21578.835,E2 -21578.835} C_VEL
LIN {X 0,Y 204.379,Z 177.112,A -85,B 0,C 180,E1 -21579.361,E2 -21579.361} C_VEL
LIN {X 0,Y 201.551,Z 175.136,A -85,B 0,C 180,E1 -21581.84,E2 -21581.84} C_VEL
LIN {X 0,Y 199.997,Z 172.374,A -85,B 0,C 180,E1 -21583.672,E2 -21583.672} C_VEL
LIN {X 0,Y 199.803,Z 171.418,A -85,B 0,C 180,E1 -21584.703,E2 -21584.703} C_VEL
LIN {X 0,Y 200.024,Z 171.173,A -85,B 0,C 180,E1 -21589.882,E2 -21589.882} C_VEL
LIN {X 0,Y 200.008,Z 171.187,A -85,B 0,C 180,E1 -21593.949,E2 -21593.949} C_VEL
LIN {X 0,Y 200.292,Z 171.127,A -85,B 0,C 180,E1 -21597.989,E2 -21597.989} C_VEL
LIN {X 0,Y 200.469,Z 171.126,A -85,B 0,C 180,E1 -21600,E2 -21600} C_VEL
LIN {X 0,Y 200.011,Z 171.161,A -85,B 0,C 180,E1 -21604.03,E2 -21604.03} C_VEL
LIN {X 0,Y 200.076,Z 171.165,A -85,B 0,C 180,E1 -21608.077,E2 -21608.077} C_VEL
LIN {X 0,Y 199.891,Z 171.204,A -85,B 0,C 180,E1 -21612.178,E2 -21612.178} C_VEL
LIN {X 0,Y 199.887,Z 171.572,A -85,B 0,C 180,E1 -21615.551,E2 -21615.551} C_VEL
LIN {X 0,Y 200.225,Z 172.868,A -85,B 0,C 180,E1 -21616.57,E2 -21616.57} C_VEL
LIN {X 0,Y 201.903,Z 175.463,A -85,B 0,C 180,E1 -21618.412,E2 -21618.412} C_VEL
LIN {X 0,Y 204.898,Z 177.56,A -85,B 0,C 180,E1 -21620.978,E2 -21620.978} C_VEL
LIN {X 0,Y 206.422,Z 180.331,A -85,B 0,C 180,E1 -21622.302,E2 -21622.302} C_VEL
LIN {X 0,Y 209.051,Z 182.678,A -85,B 0,C 180,E1 -21624.187,E2 -21624.187} C_VEL
LIN {X 0,Y 209.717,Z 183.224,A -85,B 0,C 180,E1 -21624.633,E2 -21624.633} C_VEL
LIN {X 0,Y 211.916,Z 186.564,A -85,B 0,C 180,E1 -21626.149,E2 -21626.149} C_VEL
LIN {X 0,Y 214.061,Z 188.579,A -85,B 0,C 180,E1 -21627.437,E2 -21627.437} C_VEL
LIN {X 0,Y 216.676,Z 192.182,A -85,B 0,C 180,E1 -21628.98,E2 -21628.98} C_VEL
LIN {X 0,Y 218.218,Z 193.876,A -85,B 0,C 180,E1 -21629.811,E2 -21629.811} C_VEL
LIN {X 0,Y 221.212,Z 197.686,A -85,B 0,C 180,E1 -21631.369,E2 -21631.369} C_VEL
LIN {X 0,Y 221.924,Z 198.818,A -85,B 0,C 180,E1 -21631.737,E2 -21631.737} C_VEL
LIN {X 0,Y 223.937,Z 202.613,A -85,B 0,C 180,E1 -21632.779,E2 -21632.779} C_VEL
LIN {X 0,Y 226.533,Z 210.342,A -85,B 0,C 180,E1 -21634.213,E2 -21634.213} C_VEL
LIN {X 0,Y 229.557,Z 220.098,A -85,B 0,C 180,E1 -21635.819,E2 -21635.819} C_VEL
LIN {X 0,Y 230.842,Z 223.057,A -85,B 0,C 180,E1 -21636.41,E2 -21636.41} C_VEL
LIN {X 0,Y 237.255,Z 235.65,A -85,B 0,C 180,E1 -21639.053,E2 -21639.053} C_VEL
LIN {X 0,Y 242.525,Z 247.336,A -85,B 0,C 180,E1 -21641.079,E2 -21641.079} C_VEL
LIN {X 0,Y 243.989,Z 250.954,A -85,B 0,C 180,E1 -21641.629,E2 -21641.629} C_VEL
LIN {X 0,Y 238.805,Z 331.027,A -85,B 0,C 180,E1 -21643.784,E2 -21643.784} C_VEL
LIN {X 0,Y 237.034,Z 346.001,A -85,B 0,C 180,E1 -21644.408,E2 -21644.408} C_VEL
LIN {X 0,Y 234.491,Z 360.072,A -85,B 0,C 180,E1 -21645.225,E2 -21645.225} C_VEL
LIN {X 0,Y 231.379,Z 373.615,A -85,B 0,C 180,E1 -21646.289,E2 -21646.289} C_VEL
LIN {X 0,Y 227.582,Z 387.779,A -85,B 0,C 180,E1 -21647.789,E2 -21647.789} C_VEL
LIN {X 0,Y 223.388,Z 400.832,A -85,B 0,C 180,E1 -21649.542,E2 -21649.542} C_VEL
LIN {X 0,Y 218.477,Z 413.882,A -85,B 0,C 180,E1 -21651.739,E2 -21651.739} C_VEL
LIN {X 0,Y 213.547,Z 425.693,A -85,B 0,C 180,E1 -21654.256,E2 -21654.256} C_VEL
LIN {X 0,Y 209.062,Z 435.63,A -85,B 0,C 180,E1 -21656.888,E2 -21656.888} C_VEL
LIN {X 0,Y 204.538,Z 445.354,A -85,B 0,C 180,E1 -21660.117,E2 -21660.117} C_VEL
LIN {X 0,Y 200.465,Z 453.465,A -85,B 0,C 180,E1 -21663.449,E2 -21663.449} C_VEL
LIN {X 0,Y 197.11,Z 460.173,A -85,B 0,C 180,E1 -21666.908,E2 -21666.908} C_VEL
LIN {X 0,Y 194.218,Z 466.366,A -85,B 0,C 180,E1 -21670.993,E2 -21670.993} C_VEL
LIN {X 0,Y 192.081,Z 471.155,A -85,B 0,C 180,E1 -21675.16,E2 -21675.16} C_VEL
LIN {X 0,Y 190.802,Z 474.663,A -85,B 0,C 180,E1 -21679.387,E2 -21679.387} C_VEL
LIN {X 0,Y 190.195,Z 476.97,A -85,B 0,C 180,E1 -21683.635,E2 -21683.635} C_VEL
LIN {X 0,Y 190.066,Z 478.129,A -85,B 0,C 180,E1 -21687.881,E2 -21687.881} C_VEL
LIN {X 0,Y 190.148,Z 478.281,A -85,B 0,C 180,E1 -21690,E2 -21690} C_VEL
LIN {X 0,Y 190.084,Z 477.675,A -85,B 0,C 180,E1 -21694.241,E2 -21694.241} C_VEL
LIN {X 0,Y 190.432,Z 475.927,A -85,B 0,C 180,E1 -21698.489,E2 -21698.489} C_VEL
LIN {X 0,Y 191.31,Z 473.011,A -85,B 0,C 180,E1 -21702.733,E2 -21702.733} C_VEL
LIN {X 0,Y 193.077,Z 468.861,A -85,B 0,C 180,E1 -21706.93,E2 -21706.93} C_VEL
LIN {X 0,Y 195.494,Z 463.363,A -85,B 0,C 180,E1 -21711.069,E2 -21711.069} C_VEL
LIN {X 0,Y 198.948,Z 456.372,A -85,B 0,C 180,E1 -21715.082,E2 -21715.082} C_VEL
LIN {X 0,Y 202.705,Z 448.895,A -85,B 0,C 180,E1 -21718.472,E2 -21718.472} C_VEL
LIN {X 0,Y 206.198,Z 441.463,A -85,B 0,C 180,E1 -21721.22,E2 -21721.22} C_VEL
LIN {X 0,Y 209.725,Z 433.933,A -85,B 0,C 180,E1 -21723.568,E2 -21723.568} C_VEL
LIN {X 0,Y 214.332,Z 423.698,A -85,B 0,C 180,E1 -21726.173,E2 -21726.173} C_VEL
